gfCNCPoint1[7259] = {X 558.4447, Y 7.7679, Z -1.3333, A 0.000, B 0.000, C 0.000 }
gfCNCPoint1[7260] = {X 558.1455, Y 6.8725, Z -1.3333, A 0.000, B 0.000, C 0.000 }
gfCNCPoint1[7261] = {X 558.0443, Y 5.9339, Z -1.3333, A 0.000, B 0.000, C 0.000 }
gfCNCPoint1[7262] = {X 558.0443, Y 5.0000, Z -1.3333, A 0.000, B 0.000, C 0.000 }
gfCNCPoint1[7263] = {X 558.1353, Y 4.1097, Z -1.3333, A 0.000, B 0.000, C 0.000 }
gfCNCPoint1[7264] = {X 558.4046, Y 3.2563, Z -1.3333, A 0.000, B 0.000, C 0.000 }
gfCNCPoint1[7265] = {X 558.9155, Y 2.3718, Z -1.3333, A 0.000, B 0.000, C 0.000 }
gfCNCPoint1[7266] = {X 559.6165, Y 1.6290, Z -1.3333, A 0.000, B 0.000, C 0.000 }
gfCNCPoint1[7267] = {X 560.4700, Y 1.0678, Z -1.3333, A 0.000, B 0.000, C 0.000 }
gfCNCPoint1[7268] = {X 561.4298, Y 0.7186, Z -1.3333, A 0.000, B 0.000, C 0.000 }
gfCNCPoint1[7269] = {X 562.4443, Y 0.6000, Z -1.3333, A 0.000, B 0.000, C 0.000 }
gfCNCPoint1[7270] = {X 570.9376, Y 0.6000, Z -1.3333, A 0.000, B 0.000, C 0.000 }
gfCNCPoint1[7271] = {X 571.9521, Y 0.7186, Z -1.3333, A 0.000, B 0.000, C 0.000 }
gfCNCPoint1[7272] = {X 572.9119, Y 1.0678, Z -1.3333, A 0.000, B 0.000, C 0.000 }
gfCNCPoint1[7273] = {X 573.7653, Y 1.6290, Z -1.3333, A 0.000, B 0.000, C 0.000 }
gfCNCPoint1[7274] = {X 574.4664, Y 2.3718, Z -1.3333, A 0.000, B 0.000, C 0.000 }
gfCNCPoint1[7275] = {X 574.9773, Y 3.2563, Z -1.3333, A 0.000, B 0.000, C 0.000 }
gfCNCPoint1[7276] = {X 575.2317, Y 4.0408, Z -1.3333, A 0.000, B 0.000, C 0.000 }
gfCNCPoint1[7277] = {X 575.3353, Y 4.8590, Z -1.3333, A 0.000, B 0.000, C 0.000 }
gfCNCPoint1[7278] = {X 580.1328, Y 4.7051, Z -1.3333, A 0.000, B 0.000, C 0.000 }
gfCNCPoint1[7279] = {X 580.1364, Y 4.8525, Z -1.3333, A 0.000, B 0.000, C 0.000 }
gfCNCPoint1[7280] = {X 580.1376, Y 5.0000, Z -1.3333, A 0.000, B 0.000, C 0.000 }
gfCNCPoint1[7281] = {X 580.1376, Y 5.9338, Z -1.3333, A 0.000, B 0.000, C 0.000 }
gfCNCPoint1[7282] = {X 580.0685, Y 7.0592, Z -1.3333, A 0.000, B 0.000, C 0.000 }
gfCNCPoint1[7283] = {X 579.8623, Y 8.1677, Z -1.3333, A 0.000, B 0.000, C 0.000 }
gfCNCPoint1[7284] = {X 581.2004, Y 11.4539, Z -1.3333, A 0.000, B 0.000, C 0.000 }
gfCNCPoint1[7285] = {X 582.6186, Y 7.9855, Z -1.3333, A 0.000, B 0.000, C 0.000 }
gfCNCPoint1[7286] = {X 582.4489, Y 6.9999, Z -1.3333, A 0.000, B 0.000, C 0.000 }
gfCNCPoint1[7287] = {X 582.3872, Y 6.0018, Z -1.3333, A 0.000, B 0.000, C 0.000 }
gfCNCPoint1[7288] = {X 582.3870, Y 5.0000, Z -1.3333, A 0.000, B 0.000, C 0.000 }
gfCNCPoint1[7289] = {X 582.3881, Y 4.8525, Z -1.3333, A 0.000, B 0.000, C 0.000 }
gfCNCPoint1[7290] = {X 582.3917, Y 4.7051, Z -1.3333, A 0.000, B 0.000, C 0.000 }
gfCNCPoint1[7291] = {X 580.1328, Y 4.7051, Z -1.3333, A 0.000, B 0.000, C 0.000 }
gfCNCPoint1[7292] = {X 577.7341, Y 4.7820, Z -1.3333, A 0.000, B 0.000, C 0.000 }
gfCNCPoint1[7293] = {X 577.7367, Y 4.8910, Z -1.3333, A 0.000, B 0.000, C 0.000 }
gfCNCPoint1[7294] = {X 577.7376, Y 5.0000, Z -1.3333, A 0.000, B 0.000, C 0.000 }
gfCNCPoint1[7295] = {X 577.7376, Y 5.9339, Z -1.3333, A 0.000, B 0.000, C 0.000 }
gfCNCPoint1[7296] = {X 577.6317, Y 7.1291, Z -1.3333, A 0.000, B 0.000, C 0.000 }
gfCNCPoint1[7297] = {X 577.3175, Y 8.2871, Z -1.3333, A 0.000, B 0.000, C 0.000 }
gfCNCPoint1[7298] = {X 577.5051, Y 8.7428, Z -1.3333, A 0.000, B 0.000, C 0.000 }
gfCNCPoint1[7299] = {X 581.1958, Y 17.8065, Z -1.3333, A 0.000, B 0.000, C 0.000 }
gfCNCPoint1[7300] = {X 585.1518, Y 8.1314, Z -1.3333, A 0.000, B 0.000, C 0.000 }
gfCNCPoint1[7301] = {X 584.8835, Y 7.0761, Z -1.3333, A 0.000, B 0.000, C 0.000 }
gfCNCPoint1[7302] = {X 584.7872, Y 5.9914, Z -1.3333, A 0.000, B 0.000, C 0.000 }
gfCNCPoint1[7303] = {X 584.7870, Y 5.0000, Z -1.3333, A 0.000, B 0.000, C 0.000 }
gfCNCPoint1[7304] = {X 584.7878, Y 4.8910, Z -1.3333, A 0.000, B 0.000, C 0.000 }
gfCNCPoint1[7305] = {X 584.7904, Y 4.7820, Z -1.3333, A 0.000, B 0.000, C 0.000 }
gfCNCPoint1[7306] = {X 584.9505, Y 3.5175, Z -1.3333, A 0.000, B 0.000, C 0.000 }
gfCNCPoint1[7307] = {X 585.3438, Y 2.3051, Z -1.3333, A 0.000, B 0.000, C 0.000 }
gfCNCPoint1[7308] = {X 577.1808, Y 2.3051, Z -1.3333, A 0.000, B 0.000, C 0.000 }
gfCNCPoint1[7309] = {X 577.5740, Y 3.5175, Z -1.3333, A 0.000, B 0.000, C 0.000 }
gfCNCPoint1[7310] = {X 577.7341, Y 4.7820, Z -1.3333, A 0.000, B 0.000, C 0.000 }
gfCNCPoint1[7311] = {X 575.3353, Y 4.8590, Z -1.3333, A 0.000, B 0.000, C 0.000 }
gfCNCPoint1[7312] = {X 575.3370, Y 4.9295, Z -1.3333, A 0.000, B 0.000, C 0.000 }
gfCNCPoint1[7313] = {X 575.3376, Y 5.0000, Z -1.3333, A 0.000, B 0.000, C 0.000 }
gfCNCPoint1[7314] = {X 575.3372, Y 5.9910, Z -1.3333, A 0.000, B 0.000, C 0.000 }
gfCNCPoint1[7315] = {X 575.2576, Y 6.7693, Z -1.3333, A 0.000, B 0.000, C 0.000 }
gfCNCPoint1[7316] = {X 575.0414, Y 7.5211, Z -1.3333, A 0.000, B 0.000, C 0.000 }
gfCNCPoint1[7317] = {X 574.6954, Y 8.2228, Z -1.3333, A 0.000, B 0.000, C 0.000 }
gfCNCPoint1[7318] = {X 575.2866, Y 9.6583, Z -1.3333, A 0.000, B 0.000, C 0.000 }
gfCNCPoint1[7319] = {X 578.9730, Y 18.7116, Z -1.3333, A 0.000, B 0.000, C 0.000 }
gfCNCPoint1[7320] = {X 580.9325, Y 23.5237, Z -1.3333, A 0.000, B 0.000, C 0.000 }
gfCNCPoint1[7321] = {X 581.1912, Y 24.1591, Z -1.3333, A 0.000, B 0.000, C 0.000 }
gfCNCPoint1[7322] = {X 587.7573, Y 8.1005, Z -1.3333, A 0.000, B 0.000, C 0.000 }
gfCNCPoint1[7323] = {X 587.4436, Y 7.4147, Z -1.3333, A 0.000, B 0.000, C 0.000 }
gfCNCPoint1[7324] = {X 587.2516, Y 6.6853, Z -1.3333, A 0.000, B 0.000, C 0.000 }
gfCNCPoint1[7325] = {X 587.1870, Y 5.9339, Z -1.3333, A 0.000, B 0.000, C 0.000 }
gfCNCPoint1[7326] = {X 587.1870, Y 5.0000, Z -1.3333, A 0.000, B 0.000, C 0.000 }
gfCNCPoint1[7327] = {X 587.2780, Y 4.1097, Z -1.3333, A 0.000, B 0.000, C 0.000 }
gfCNCPoint1[7328] = {X 587.5472, Y 3.2563, Z -1.3333, A 0.000, B 0.000, C 0.000 }
gfCNCPoint1[7329] = {X 588.0581, Y 2.3718, Z -1.3333, A 0.000, B 0.000, C 0.000 }
gfCNCPoint1[7330] = {X 588.7592, Y 1.6290, Z -1.3333, A 0.000, B 0.000, C 0.000 }
gfCNCPoint1[7331] = {X 589.6126, Y 1.0678, Z -1.3333, A 0.000, B 0.000, C 0.000 }
gfCNCPoint1[7332] = {X 590.5725, Y 0.7186, Z -1.3333, A 0.000, B 0.000, C 0.000 }
gfCNCPoint1[7333] = {X 591.5870, Y 0.6000, Z -1.3333, A 0.000, B 0.000, C 0.000 }
gfCNCPoint1[7334] = {X 600.0000, Y 0.6000, Z -1.3333, A 0.000, B 0.000, C 0.000 }
gfCNCPoint1[7335] = {X 600.8720, Y 0.6873, Z -1.3333, A 0.000, B 0.000, C 0.000 }
gfCNCPoint1[7336] = {X 601.7093, Y 0.9456, Z -1.3333, A 0.000, B 0.000, C 0.000 }
gfCNCPoint1[7337] = {X 602.4789, Y 1.3648, Z -1.3333, A 0.000, B 0.000, C 0.000 }
gfCNCPoint1[7338] = {X 603.1502, Y 1.9281, Z -1.3333, A 0.000, B 0.000, C 0.000 }
gfCNCPoint1[7339] = {X 603.6965, Y 2.6133, Z -1.3333, A 0.000, B 0.000, C 0.000 }
gfCNCPoint1[7340] = {X 603.6965, Y 1.8140, Z -1.3333, A 0.000, B 0.000, C 0.000 }
gfCNCPoint1[7341] = {X 602.9511, Y 1.1135, Z -1.3333, A 0.000, B 0.000, C 0.000 }
gfCNCPoint1[7342] = {X 602.0762, Y 0.5837, Z -1.3333, A 0.000, B 0.000, C 0.000 }
gfCNCPoint1[7343] = {X 601.1100, Y 0.2479, Z -1.3333, A 0.000, B 0.000, C 0.000 }
gfCNCPoint1[7344] = {X 600.0950, Y 0.1209, Z -1.3333, A 0.000, B 0.000, C 0.000 }
gfCNCPoint1[7345] = {X 600.0947, Y -0.0187, Z -1.3333, A 0.000, B 0.000, C 0.000 }
gfCNCPoint1[7346] = {X 600.0671, Y -0.0697, Z -1.3333, A 0.000, B 0.000, C 0.000 }
gfCNCPoint1[7347] = {X 600.0148, Y -0.0949, Z -1.3333, A 0.000, B 0.000, C 0.000 }
gfCNCPoint1[7348] = {X 351.5614, Y -0.0949, Z -1.3333, A 0.000, B 0.000, C 0.000 }
gfCNCPoint1[7349] = {X 351.4045, Y -0.1238, Z -1.3333, A 0.000, B 0.000, C 0.000 }
gfCNCPoint1[7350] = {X 348.9100, Y -0.4700, Z -1.3333, A 0.000, B 0.000, C 0.000 }
gfCNCPoint1[7351] = {X 346.3941, Y -0.5809, Z -1.3333, A 0.000, B 0.000, C 0.000 }
gfCNCPoint1[7352] = {X 343.8788, Y -0.4555, Z -1.3333, A 0.000, B 0.000, C 0.000 }
gfCNCPoint1[7353] = {X 341.3863, Y -0.0949, Z -1.3333, A 0.000, B 0.000, C 0.000 }
gfCNCPoint1[7354] = {X -0.0148, Y -0.0949, Z -1.3333, A 0.000, B 0.000, C 0.000 }
gfCNCPoint1[7355] = {X -0.0671, Y -0.0697, Z -1.3333, A 0.000, B 0.000, C 0.000 }
gfCNCPoint1[7356] = {X -0.0947, Y -0.0187, Z -1.3333, A 0.000, B 0.000, C 0.000 }
gfCNCPoint1[7357] = {X -0.0965, Y 0.8569, Z -1.3333, A 0.000, B 0.000, C 0.000 }
gfCNCPoint1[7358] = {X -0.0965, Y 8.7890, Z -1.3333, A 0.000, B 0.000, C 0.000 }
gfCNCPoint1[7359] = {X -0.7633, Y 8.9979, Z -1.3333, A 0.000, B 0.000, C 0.000 }
gfCNCPoint1[7360] = {X -1.3935, Y 9.2998, Z -1.3333, A 0.000, B 0.000, C 0.000 }
gfCNCPoint1[7361] = {X -1.9904, Y 9.6404, Z -1.3333, A 0.000, B 0.000, C 0.000 }
gfCNCPoint1[7362] = {X -2.6454, Y 10.0884, Z -1.3333, A 0.000, B 0.000, C 0.000 }
gfCNCPoint1[7363] = {X -3.2192, Y 10.6366, Z -1.3333, A 0.000, B 0.000, C 0.000 }
gfCNCPoint1[7364] = {X -3.6965, Y 11.2705, Z -1.3333, A 0.000, B 0.000, C 0.000 }
gfCNCPoint1[7365] = {X -3.6965, Y 12.3459, Z -1.3333, A 0.000, B 0.000, C 0.000 }
gfCNCPoint1[7366] = {X -3.2331, Y 11.4382, Z -1.3333, A 0.000, B 0.000, C 0.000 }
gfCNCPoint1[7367] = {X -2.5733, Y 10.6615, Z -1.3333, A 0.000, B 0.000, C 0.000 }
gfCNCPoint1[7368] = {X -1.7526, Y 10.0573, Z -1.3333, A 0.000, B 0.000, C 0.000 }
gfCNCPoint1[7369] = {X -1.0994, Y 9.6852, Z -1.3333, A 0.000, B 0.000, C 0.000 }
gfCNCPoint1[7370] = {X -0.1607, Y 9.3012, Z -1.3333, A 0.000, B 0.000, C 0.000 }
gfCNCPoint1[7371] = {X 0.8409, Y 9.1423, Z -1.3333, A 0.000, B 0.000, C 0.000 }
gfCNCPoint1[7372] = {X 1.8523, Y 9.2169, Z -1.3333, A 0.000, B 0.000, C 0.000 }
gfCNCPoint1[7373] = {X 2.2372, Y 9.3088, Z -1.3333, A 0.000, B 0.000, C 0.000 }
gfCNCPoint1[7374] = {X 2.6123, Y 9.4348, Z -1.3333, A 0.000, B 0.000, C 0.000 }
gfCNCPoint1[7375] = {X 3.3801, Y 9.0795, Z -1.3333, A 0.000, B 0.000, C 0.000 }
gfCNCPoint1[7376] = {X 4.1677, Y 8.7704, Z -1.3333, A 0.000, B 0.000, C 0.000 }
gfCNCPoint1[7377] = {X 6.0851, Y 8.0995, Z -1.3333, A 0.000, B 0.000, C 0.000 }
gfCNCPoint1[7378] = {X 8.0532, Y 7.5963, Z -1.3333, A 0.000, B 0.000, C 0.000 }
gfCNCPoint1[7379] = {X 10.0574, Y 7.2648, Z -1.3333, A 0.000, B 0.000, C 0.000 }
gfCNCPoint1[7380] = {X 12.0827, Y 7.1073, Z -1.3333, A 0.000, B 0.000, C 0.000 }
gfCNCPoint1[7381] = {X 14.1141, Y 7.1249, Z -1.3333, A 0.000, B 0.000, C 0.000 }
gfCNCPoint1[7382] = {X 16.1363, Y 7.3177, Z -1.3333, A 0.000, B 0.000, C 0.000 }
gfCNCPoint1[7383] = {X 16.5409, Y 7.3732, Z -1.3333, A 0.000, B 0.000, C 0.000 }
gfCNCPoint1[7384] = {X 18.2850, Y 7.7308, Z -1.3333, A 0.000, B 0.000, C 0.000 }
gfCNCPoint1[7385] = {X 19.9840, Y 8.2634, Z -1.3333, A 0.000, B 0.000, C 0.000 }
gfCNCPoint1[7386] = {X 21.6202, Y 8.9655, Z -1.3333, A 0.000, B 0.000, C 0.000 }
gfCNCPoint1[7387] = {X 23.1768, Y 9.8298, Z -1.3333, A 0.000, B 0.000, C 0.000 }
gfCNCPoint1[7388] = {X 24.6377, Y 10.8475, Z -1.3333, A 0.000, B 0.000, C 0.000 }
gfCNCPoint1[7389] = {X 25.7295, Y 11.8031, Z -1.3333, A 0.000, B 0.000, C 0.000 }
gfCNCPoint1[7390] = {X 26.7088, Y 12.8735, Z -1.3333, A 0.000, B 0.000, C 0.000 }
gfCNCPoint1[7391] = {X 27.5636, Y 14.0458, Z -1.3333, A 0.000, B 0.000, C 0.000 }
gfCNCPoint1[7392] = {X 28.2836, Y 15.3054, Z -1.3333, A 0.000, B 0.000, C 0.000 }
gfCNCPoint1[7393] = {X 28.8598, Y 16.6369, Z -1.3333, A 0.000, B 0.000, C 0.000 }
gfCNCPoint1[7394] = {X 29.3358, Y 18.3014, Z -1.3333, A 0.000, B 0.000, C 0.000 }
gfCNCPoint1[7395] = {X 29.6183, Y 20.0095, Z -1.3333, A 0.000, B 0.000, C 0.000 }
gfCNCPoint1[7396] = {X 29.7035, Y 21.7387, Z -1.3333, A 0.000, B 0.000, C 0.000 }
gfCNCPoint1[7397] = {X 29.5903, Y 23.4663, Z -1.3333, A 0.000, B 0.000, C 0.000 }
gfCNCPoint1[7398] = {X 29.2802, Y 25.1696, Z -1.3333, A 0.000, B 0.000, C 0.000 }
gfCNCPoint1[7399] = {X 28.7891, Y 26.7453, Z -1.3333, A 0.000, B 0.000, C 0.000 }
gfCNCPoint1[7400] = {X 28.0825, Y 28.2367, Z -1.3333, A 0.000, B 0.000, C 0.000 }
gfCNCPoint1[7401] = {X 27.1741, Y 29.6147, Z -1.3333, A 0.000, B 0.000, C 0.000 }
gfCNCPoint1[7402] = {X 26.3570, Y 30.5719, Z -1.3333, A 0.000, B 0.000, C 0.000 }
gfCNCPoint1[7403] = {X 25.4424, Y 31.4364, Z -1.3333, A 0.000, B 0.000, C 0.000 }
gfCNCPoint1[7404] = {X 25.6930, Y 31.5320, Z -1.3333, A 0.000, B 0.000, C 0.000 }
gfCNCPoint1[7405] = {X 25.9374, Y 31.6427, Z -1.3333, A 0.000, B 0.000, C 0.000 }
gfCNCPoint1[7406] = {X 26.6622, Y 32.0899, Z -1.3333, A 0.000, B 0.000, C 0.000 }
gfCNCPoint1[7407] = {X 27.2873, Y 32.6684, Z -1.3333, A 0.000, B 0.000, C 0.000 }
gfCNCPoint1[7408] = {X 27.6590, Y 33.1492, Z -1.3333, A 0.000, B 0.000, C 0.000 }
gfCNCPoint1[7409] = {X 27.9609, Y 33.6766, Z -1.3333, A 0.000, B 0.000, C 0.000 }
gfCNCPoint1[7410] = {X 30.9820, Y 39.9182, Z -1.3333, A 0.000, B 0.000, C 0.000 }
gfCNCPoint1[7411] = {X 31.3085, Y 40.8441, Z -1.3333, A 0.000, B 0.000, C 0.000 }
gfCNCPoint1[7412] = {X 31.4215, Y 41.8194, Z -1.3333, A 0.000, B 0.000, C 0.000 }
gfCNCPoint1[7413] = {X 31.3155, Y 42.7955, Z -1.3333, A 0.000, B 0.000, C 0.000 }
gfCNCPoint1[7414] = {X 30.9956, Y 43.7238, Z -1.3333, A 0.000, B 0.000, C 0.000 }
gfCNCPoint1[7415] = {X 30.4779, Y 44.5580, Z -1.3333, A 0.000, B 0.000, C 0.000 }
gfCNCPoint1[7416] = {X 29.7880, Y 45.2567, Z -1.3333, A 0.000, B 0.000, C 0.000 }
gfCNCPoint1[7417] = {X 29.2515, Y 45.6905, Z -1.3333, A 0.000, B 0.000, C 0.000 }
gfCNCPoint1[7418] = {X 28.5397, Y 46.1587, Z -1.3333, A 0.000, B 0.000, C 0.000 }
gfCNCPoint1[7419] = {X 27.7513, Y 46.4816, Z -1.3333, A 0.000, B 0.000, C 0.000 }
gfCNCPoint1[7420] = {X 26.9155, Y 46.6472, Z -1.3333, A 0.000, B 0.000, C 0.000 }
gfCNCPoint1[7421] = {X 26.0635, Y 46.6494, Z -1.3333, A 0.000, B 0.000, C 0.000 }
gfCNCPoint1[7422] = {X 25.2269, Y 46.4880, Z -1.3333, A 0.000, B 0.000, C 0.000 }
gfCNCPoint1[7423] = {X 23.2106, Y 47.5426, Z -1.3333, A 0.000, B 0.000, C 0.000 }
gfCNCPoint1[7424] = {X 21.1166, Y 48.4331, Z -1.3333, A 0.000, B 0.000, C 0.000 }
gfCNCPoint1[7425] = {X 18.9583, Y 49.1538, Z -1.3333, A 0.000, B 0.000, C 0.000 }
gfCNCPoint1[7426] = {X 18.4672, Y 49.2899, Z -1.3333, A 0.000, B 0.000, C 0.000 }
gfCNCPoint1[7427] = {X 16.5967, Y 49.7226, Z -1.3333, A 0.000, B 0.000, C 0.000 }
gfCNCPoint1[7428] = {X 14.6960, Y 49.9931, Z -1.3333, A 0.000, B 0.000, C 0.000 }
gfCNCPoint1[7429] = {X 12.7791, Y 50.0995, Z -1.3333, A 0.000, B 0.000, C 0.000 }
gfCNCPoint1[7430] = {X 10.8601, Y 50.0409, Z -1.3333, A 0.000, B 0.000, C 0.000 }
gfCNCPoint1[7431] = {X 8.9532, Y 49.8178, Z -1.3333, A 0.000, B 0.000, C 0.000 }
gfCNCPoint1[7432] = {X 8.2283, Y 49.7011, Z -1.3333, A 0.000, B 0.000, C 0.000 }
gfCNCPoint1[7433] = {X 6.5700, Y 49.3105, Z -1.3333, A 0.000, B 0.000, C 0.000 }
gfCNCPoint1[7434] = {X 4.9585, Y 48.7578, Z -1.3333, A 0.000, B 0.000, C 0.000 }
gfCNCPoint1[7435] = {X 3.4094, Y 48.0486, Z -1.3333, A 0.000, B 0.000, C 0.000 }
gfCNCPoint1[7436] = {X 2.3355, Y 47.4411, Z -1.3333, A 0.000, B 0.000, C 0.000 }
gfCNCPoint1[7437] = {X 1.3077, Y 46.7583, Z -1.3333, A 0.000, B 0.000, C 0.000 }
gfCNCPoint1[7438] = {X -0.0256, Y 45.6860, Z -1.3333, A 0.000, B 0.000, C 0.000 }
gfCNCPoint1[7439] = {X -1.2107, Y 44.4520, Z -1.3333, A 0.000, B 0.000, C 0.000 }
gfCNCPoint1[7440] = {X -2.2282, Y 43.0765, Z -1.3333, A 0.000, B 0.000, C 0.000 }
gfCNCPoint1[7441] = {X -3.0614, Y 41.5820, Z -1.3333, A 0.000, B 0.000, C 0.000 }
gfCNCPoint1[7442] = {X -3.6965, Y 39.9933, Z -1.3333, A 0.000, B 0.000, C 0.000 }
gfCNCPoint1[7443] = {X -3.6965, Y 41.3449, Z -1.3333, A 0.000, B 0.000, C 0.000 }
gfCNCPoint1[7444] = {X -3.0079, Y 42.7182, Z -1.3333, A 0.000, B 0.000, C 0.000 }
gfCNCPoint1[7445] = {X -2.1712, Y 44.0066, Z -1.3333, A 0.000, B 0.000, C 0.000 }
gfCNCPoint1[7446] = {X -1.1967, Y 45.1942, Z -1.3333, A 0.000, B 0.000, C 0.000 }
gfCNCPoint1[7447] = {X -0.0965, Y 46.2663, Z -1.3333, A 0.000, B 0.000, C 0.000 }
gfCNCPoint1[7448] = {X -0.0965, Y 99.1431, Z -1.3333, A 0.000, B 0.000, C 0.000 }
gfCNCPoint1[7449] = {X -0.0947, Y 100.0187, Z -1.3333, A 0.000, B 0.000, C 0.000 }
gfCNCPoint1[7450] = {X -0.0671, Y 100.0697, Z -1.3333, A 0.000, B 0.000, C 0.000 }
gfCNCPoint1[7451] = {X -0.0148, Y 100.0949, Z -1.3333, A 0.000, B 0.000, C 0.000 }
gfCNCPoint1[7452] = {X 120.5925, Y 100.0949, Z -1.3333, A 0.000, B 0.000, C 0.000 }
gfCNCPoint1[7453] = {X 121.0613, Y 100.8811, Z -1.3333, A 0.000, B 0.000, C 0.000 }
gfCNCPoint1[7454] = {X 121.6686, Y 101.5660, Z -1.3333, A 0.000, B 0.000, C 0.000 }
gfCNCPoint1[7455] = {X 122.3931, Y 102.1254, Z -1.3333, A 0.000, B 0.000, C 0.000 }
gfCNCPoint1[7456] = {X 123.2094, Y 102.5396, Z -1.3333, A 0.000, B 0.000, C 0.000 }
gfCNCPoint1[7457] = {X 124.0887, Y 102.7942, Z -1.3333, A 0.000, B 0.000, C 0.000 }
gfCNCPoint1[7458] = {X 125.0000, Y 102.8800, Z -1.3333, A 0.000, B 0.000, C 0.000 }
gfCNCPoint1[7459] = {X 143.7791, Y 102.8800, Z -1.3333, A 0.000, B 0.000, C 0.000 }
gfCNCPoint1[7460] = {X 144.6904, Y 102.7942, Z -1.3333, A 0.000, B 0.000, C 0.000 }
gfCNCPoint1[7461] = {X 145.5697, Y 102.5396, Z -1.3333, A 0.000, B 0.000, C 0.000 }
gfCNCPoint1[7462] = {X 146.3860, Y 102.1254, Z -1.3333, A 0.000, B 0.000, C 0.000 }
gfCNCPoint1[7463] = {X 147.1105, Y 101.5660, Z -1.3333, A 0.000, B 0.000, C 0.000 }
gfCNCPoint1[7464] = {X 147.7178, Y 100.8811, Z -1.3333, A 0.000, B 0.000, C 0.000 }
gfCNCPoint1[7465] = {X 148.1866, Y 100.0949, Z -1.3333, A 0.000, B 0.000, C 0.000 }
gfCNCPoint1[7466] = {X 150.8370, Y 100.0949, Z -1.3333, A 0.000, B 0.000, C 0.000 }
gfCNCPoint1[7467] = {X 150.8370, Y 95.2949, Z -1.3333, A 0.000, B 0.000, C 0.000 }
gfCNCPoint1[7468] = {X 187.9257, Y 95.2949, Z -1.3333, A 0.000, B 0.000, C 0.000 }
gfCNCPoint1[7469] = {X 187.9777, Y 95.0989, Z -1.3333, A 0.000, B 0.000, C 0.000 }
gfCNCPoint1[7470] = {X 188.0352, Y 94.9045, Z -1.3333, A 0.000, B 0.000, C 0.000 }
gfCNCPoint1[7471] = {X 187.2619, Y 94.0602, Z -1.3333, A 0.000, B 0.000, C 0.000 }
gfCNCPoint1[7472] = {X 151.4055, Y 94.0602, Z -1.3333, A 0.000, B 0.000, C 0.000 }
gfCNCPoint1[7473] = {X 150.7052, Y 94.8361, Z -1.3333, A 0.000, B 0.000, C 0.000 }
gfCNCPoint1[7474] = {X 150.7748, Y 95.0644, Z -1.3333, A 0.000, B 0.000, C 0.000 }
gfCNCPoint1[7475] = {X 150.8370, Y 95.2949, Z -1.3333, A 0.000, B 0.000, C 0.000 }
gfCNCPoint1[7476] = {X 150.8370, Y 97.6949, Z -1.3333, A 0.000, B 0.000, C 0.000 }
gfCNCPoint1[7477] = {X 190.1070, Y 97.6949, Z -1.3333, A 0.000, B 0.000, C 0.000 }
gfCNCPoint1[7478] = {X 190.1070, Y 97.0659, Z -1.3333, A 0.000, B 0.000, C 0.000 }
gfCNCPoint1[7479] = {X 190.1938, Y 96.1495, Z -1.3333, A 0.000, B 0.000, C 0.000 }
gfCNCPoint1[7480] = {X 190.4511, Y 95.2657, Z -1.3333, A 0.000, B 0.000, C 0.000 }
gfCNCPoint1[7481] = {X 190.8699, Y 94.4460, Z -1.3333, A 0.000, B 0.000, C 0.000 }
gfCNCPoint1[7482] = {X 188.3182, Y 91.6602, Z -1.3333, A 0.000, B 0.000, C 0.000 }
gfCNCPoint1[7483] = {X 150.3387, Y 91.6602, Z -1.3333, A 0.000, B 0.000, C 0.000 }
gfCNCPoint1[7484] = {X 147.8631, Y 94.4029, Z -1.3333, A 0.000, B 0.000, C 0.000 }
gfCNCPoint1[7485] = {X 148.2972, Y 95.2330, Z -1.3333, A 0.000, B 0.000, C 0.000 }
gfCNCPoint1[7486] = {X 148.5657, Y 96.1303, Z -1.3333, A 0.000, B 0.000, C 0.000 }
gfCNCPoint1[7487] = {X 148.6591, Y 97.0623, Z -1.3333, A 0.000, B 0.000, C 0.000 }
gfCNCPoint1[7488] = {X 148.6591, Y 97.6949, Z -1.3333, A 0.000, B 0.000, C 0.000 }
gfCNCPoint1[7489] = {X 150.8370, Y 97.6949, Z -1.3333, A 0.000, B 0.000, C 0.000 }
gfCNCPoint1[7490] = {X 150.8370, Y 100.0949, Z -1.3333, A 0.000, B 0.000, C 0.000 }
gfCNCPoint1[7491] = {X 190.5795, Y 100.0949, Z -1.3333, A 0.000, B 0.000, C 0.000 }
gfCNCPoint1[7492] = {X 191.0482, Y 100.8811, Z -1.3333, A 0.000, B 0.000, C 0.000 }
gfCNCPoint1[7493] = {X 191.6556, Y 101.5660, Z -1.3333, A 0.000, B 0.000, C 0.000 }
gfCNCPoint1[7494] = {X 192.3801, Y 102.1254, Z -1.3333, A 0.000, B 0.000, C 0.000 }
gfCNCPoint1[7495] = {X 193.1964, Y 102.5396, Z -1.3333, A 0.000, B 0.000, C 0.000 }
gfCNCPoint1[7496] = {X 194.0756, Y 102.7942, Z -1.3333, A 0.000, B 0.000, C 0.000 }
gfCNCPoint1[7497] = {X 194.9870, Y 102.8800, Z -1.3333, A 0.000, B 0.000, C 0.000 }
gfCNCPoint1[7498] = {X 212.6141, Y 102.8800, Z -1.3333, A 0.000, B 0.000, C 0.000 }
gfCNCPoint1[7499] = {X 213.0066, Y 102.8642, Z -1.3333, A 0.000, B 0.000, C 0.000 }
gfCNCPoint1[7500] = {X 213.3966, Y 102.8169, Z -1.3333, A 0.000, B 0.000, C 0.000 }
gfCNCPoint1[7501] = {X 213.7865, Y 102.8642, Z -1.3333, A 0.000, B 0.000, C 0.000 }
gfCNCPoint1[7502] = {X 214.1790, Y 102.8800, Z -1.3333, A 0.000, B 0.000, C 0.000 }
gfCNCPoint1[7503] = {X 233.4798, Y 102.8800, Z -1.3333, A 0.000, B 0.000, C 0.000 }
gfCNCPoint1[7504] = {X 234.3911, Y 102.7942, Z -1.3333, A 0.000, B 0.000, C 0.000 }
gfCNCPoint1[7505] = {X 235.2704, Y 102.5396, Z -1.3333, A 0.000, B 0.000, C 0.000 }
gfCNCPoint1[7506] = {X 236.0866, Y 102.1254, Z -1.3333, A 0.000, B 0.000, C 0.000 }
gfCNCPoint1[7507] = {X 236.8112, Y 101.5660, Z -1.3333, A 0.000, B 0.000, C 0.000 }
gfCNCPoint1[7508] = {X 237.4185, Y 100.8811, Z -1.3333, A 0.000, B 0.000, C 0.000 }
gfCNCPoint1[7509] = {X 237.8873, Y 100.0949, Z -1.3333, A 0.000, B 0.000, C 0.000 }
gfCNCPoint1[7510] = {X 261.4765, Y 100.0949, Z -1.3333, A 0.000, B 0.000, C 0.000 }
gfCNCPoint1[7511] = {X 261.4765, Y 90.4949, Z -1.3333, A 0.000, B 0.000, C 0.000 }
gfCNCPoint1[7512] = {X 266.0962, Y 90.4949, Z -1.3333, A 0.000, B 0.000, C 0.000 }
gfCNCPoint1[7513] = {X 266.1752, Y 90.3746, Z -1.3333, A 0.000, B 0.000, C 0.000 }
gfCNCPoint1[7514] = {X 266.2556, Y 90.2554, Z -1.3333, A 0.000, B 0.000, C 0.000 }
gfCNCPoint1[7515] = {X 263.5087, Y 89.1786, Z -1.3333, A 0.000, B 0.000, C 0.000 }
gfCNCPoint1[7516] = {X 261.4765, Y 90.4949, Z -1.3333, A 0.000, B 0.000, C 0.000 }
gfCNCPoint1[7517] = {X 261.4765, Y 92.8949, Z -1.3333, A 0.000, B 0.000, C 0.000 }
gfCNCPoint1[7518] = {X 267.4974, Y 92.8949, Z -1.3333, A 0.000, B 0.000, C 0.000 }
gfCNCPoint1[7519] = {X 267.8429, Y 92.2375, Z -1.3333, A 0.000, B 0.000, C 0.000 }
gfCNCPoint1[7520] = {X 268.2378, Y 91.6085, Z -1.3333, A 0.000, B 0.000, C 0.000 }
gfCNCPoint1[7521] = {X 269.1700, Y 90.4463, Z -1.3333, A 0.000, B 0.000, C 0.000 }
gfCNCPoint1[7522] = {X 270.2694, Y 89.4409, Z -1.3333, A 0.000, B 0.000, C 0.000 }
gfCNCPoint1[7523] = {X 270.2694, Y 89.2510, Z -1.3333, A 0.000, B 0.000, C 0.000 }
gfCNCPoint1[7524] = {X 263.2378, Y 86.4946, Z -1.3333, A 0.000, B 0.000, C 0.000 }
gfCNCPoint1[7525] = {X 253.3566, Y 92.8949, Z -1.3333, A 0.000, B 0.000, C 0.000 }
gfCNCPoint1[7526] = {X 261.4765, Y 92.8949, Z -1.3333, A 0.000, B 0.000, C 0.000 }
gfCNCPoint1[7527] = {X 261.4765, Y 95.2949, Z -1.3333, A 0.000, B 0.000, C 0.000 }
gfCNCPoint1[7528] = {X 269.1714, Y 95.2949, Z -1.3333, A 0.000, B 0.000, C 0.000 }
gfCNCPoint1[7529] = {X 269.5516, Y 94.1744, Z -1.3333, A 0.000, B 0.000, C 0.000 }
gfCNCPoint1[7530] = {X 270.1083, Y 93.1302, Z -1.3333, A 0.000, B 0.000, C 0.000 }
gfCNCPoint1[7531] = {X 270.8267, Y 92.1901, Z -1.3333, A 0.000, B 0.000, C 0.000 }
gfCNCPoint1[7532] = {X 271.6880, Y 91.3787, Z -1.3333, A 0.000, B 0.000, C 0.000 }
gfCNCPoint1[7533] = {X 272.6694, Y 90.7176, Z -1.3333, A 0.000, B 0.000, C 0.000 }
gfCNCPoint1[7534] = {X 272.6694, Y 87.6139, Z -1.3333, A 0.000, B 0.000, C 0.000 }
gfCNCPoint1[7535] = {X 262.9669, Y 83.8106, Z -1.3333, A 0.000, B 0.000, C 0.000 }
gfCNCPoint1[7536] = {X 245.2366, Y 95.2949, Z -1.3333, A 0.000, B 0.000, C 0.000 }
gfCNCPoint1[7537] = {X 261.4765, Y 95.2949, Z -1.3333, A 0.000, B 0.000, C 0.000 }
gfCNCPoint1[7538] = {X 261.4765, Y 97.6949, Z -1.3333, A 0.000, B 0.000, C 0.000 }
gfCNCPoint1[7539] = {X 271.3527, Y 97.6949, Z -1.3333, A 0.000, B 0.000, C 0.000 }
gfCNCPoint1[7540] = {X 271.3529, Y 97.0186, Z -1.3333, A 0.000, B 0.000, C 0.000 }
gfCNCPoint1[7541] = {X 271.4810, Y 95.9545, Z -1.3333, A 0.000, B 0.000, C 0.000 }
gfCNCPoint1[7542] = {X 271.8382, Y 94.9440, Z -1.3333, A 0.000, B 0.000, C 0.000 }
gfCNCPoint1[7543] = {X 272.4073, Y 94.0359, Z -1.3333, A 0.000, B 0.000, C 0.000 }
gfCNCPoint1[7544] = {X 273.1610, Y 93.2739, Z -1.3333, A 0.000, B 0.000, C 0.000 }
gfCNCPoint1[7545] = {X 274.0629, Y 92.6949, Z -1.3333, A 0.000, B 0.000, C 0.000 }
gfCNCPoint1[7546] = {X 275.0694, Y 92.3266, Z -1.3333, A 0.000, B 0.000, C 0.000 }
gfCNCPoint1[7547] = {X 275.0694, Y 85.9769, Z -1.3333, A 0.000, B 0.000, C 0.000 }
gfCNCPoint1[7548] = {X 262.6982, Y 81.1274, Z -1.3333, A 0.000, B 0.000, C 0.000 }
gfCNCPoint1[7549] = {X 262.5768, Y 81.2038, Z -1.3333, A 0.000, B 0.000, C 0.000 }
gfCNCPoint1[7550] = {X 238.3583, Y 96.8907, Z -1.3333, A 0.000, B 0.000, C 0.000 }
gfCNCPoint1[7551] = {X 238.3598, Y 97.0659, Z -1.3333, A 0.000, B 0.000, C 0.000 }
gfCNCPoint1[7552] = {X 238.3598, Y 97.6949, Z -1.3333, A 0.000, B 0.000, C 0.000 }
gfCNCPoint1[7553] = {X 261.4765, Y 97.6949, Z -1.3333, A 0.000, B 0.000, C 0.000 }
gfCNCPoint1[7554] = {X 261.4765, Y 100.0949, Z -1.3333, A 0.000, B 0.000, C 0.000 }
gfCNCPoint1[7555] = {X 271.8252, Y 100.0949, Z -1.3333, A 0.000, B 0.000, C 0.000 }
gfCNCPoint1[7556] = {X 272.2940, Y 100.8811, Z -1.3333, A 0.000, B 0.000, C 0.000 }
gfCNCPoint1[7557] = {X 272.9013, Y 101.5660, Z -1.3333, A 0.000, B 0.000, C 0.000 }
gfCNCPoint1[7558] = {X 273.6258, Y 102.1254, Z -1.3333, A 0.000, B 0.000, C 0.000 }
gfCNCPoint1[7559] = {X 274.4421, Y 102.5396, Z -1.3333, A 0.000, B 0.000, C 0.000 }
gfCNCPoint1[7560] = {X 275.3214, Y 102.7942, Z -1.3333, A 0.000, B 0.000, C 0.000 }
gfCNCPoint1[7561] = {X 276.2327, Y 102.8800, Z -1.3333, A 0.000, B 0.000, C 0.000 }
gfCNCPoint1[7562] = {X 292.7731, Y 102.8800, Z -1.3333, A 0.000, B 0.000, C 0.000 }
gfCNCPoint1[7563] = {X 293.6844, Y 102.7942, Z -1.3333, A 0.000, B 0.000, C 0.000 }
gfCNCPoint1[7564] = {X 294.5637, Y 102.5396, Z -1.3333, A 0.000, B 0.000, C 0.000 }
gfCNCPoint1[7565] = {X 295.3799, Y 102.1254, Z -1.3333, A 0.000, B 0.000, C 0.000 }
gfCNCPoint1[7566] = {X 296.1045, Y 101.5660, Z -1.3333, A 0.000, B 0.000, C 0.000 }
gfCNCPoint1[7567] = {X 296.7118, Y 100.8811, Z -1.3333, A 0.000, B 0.000, C 0.000 }
gfCNCPoint1[7568] = {X 297.1806, Y 100.0949, Z -1.3333, A 0.000, B 0.000, C 0.000 }
gfCNCPoint1[7569] = {X 319.1370, Y 100.0949, Z -1.3333, A 0.000, B 0.000, C 0.000 }
gfCNCPoint1[7570] = {X 321.4387, Y 100.8673, Z -1.3333, A 0.000, B 0.000, C 0.000 }
gfCNCPoint1[7571] = {X 323.7830, Y 101.4988, Z -1.3333, A 0.000, B 0.000, C 0.000 }
gfCNCPoint1[7572] = {X 326.1613, Y 101.9871, Z -1.3333, A 0.000, B 0.000, C 0.000 }
gfCNCPoint1[7573] = {X 329.6396, Y 102.5406, Z -1.3333, A 0.000, B 0.000, C 0.000 }
gfCNCPoint1[7574] = {X 333.1371, Y 102.9560, Z -1.3333, A 0.000, B 0.000, C 0.000 }
gfCNCPoint1[7575] = {X 336.6483, Y 103.2328, Z -1.3333, A 0.000, B 0.000, C 0.000 }
gfCNCPoint1[7576] = {X 342.8092, Y 103.5147, Z -1.3333, A 0.000, B 0.000, C 0.000 }
gfCNCPoint1[7577] = {X 348.9761, Y 103.5913, Z -1.3333, A 0.000, B 0.000, C 0.000 }
gfCNCPoint1[7578] = {X 355.1421, Y 103.4625, Z -1.3333, A 0.000, B 0.000, C 0.000 }
gfCNCPoint1[7579] = {X 361.3005, Y 103.1283, Z -1.3333, A 0.000, B 0.000, C 0.000 }
gfCNCPoint1[7580] = {X 365.1926, Y 102.7577, Z -1.3333, A 0.000, B 0.000, C 0.000 }
gfCNCPoint1[7581] = {X 369.0624, Y 102.2005, Z -1.3333, A 0.000, B 0.000, C 0.000 }
gfCNCPoint1[7582] = {X 372.9009, Y 101.4578, Z -1.3333, A 0.000, B 0.000, C 0.000 }
gfCNCPoint1[7583] = {X 375.2305, Y 100.8566, Z -1.3333, A 0.000, B 0.000, C 0.000 }
gfCNCPoint1[7584] = {X 377.5126, Y 100.0949, Z -1.3333, A 0.000, B 0.000, C 0.000 }
gfCNCPoint1[7585] = {X 391.9985, Y 100.0949, Z -1.3333, A 0.000, B 0.000, C 0.000 }
gfCNCPoint1[7586] = {X 392.4672, Y 100.8811, Z -1.3333, A 0.000, B 0.000, C 0.000 }
gfCNCPoint1[7587] = {X 393.0746, Y 101.5660, Z -1.3333, A 0.000, B 0.000, C 0.000 }
gfCNCPoint1[7588] = {X 393.7991, Y 102.1254, Z -1.3333, A 0.000, B 0.000, C 0.000 }
gfCNCPoint1[7589] = {X 394.6154, Y 102.5396, Z -1.3333, A 0.000, B 0.000, C 0.000 }
gfCNCPoint1[7590] = {X 395.4946, Y 102.7942, Z -1.3333, A 0.000, B 0.000, C 0.000 }
gfCNCPoint1[7591] = {X 396.4059, Y 102.8800, Z -1.3333, A 0.000, B 0.000, C 0.000 }
gfCNCPoint1[7592] = {X 415.7067, Y 102.8800, Z -1.3333, A 0.000, B 0.000, C 0.000 }
gfCNCPoint1[7593] = {X 416.6180, Y 102.7942, Z -1.3333, A 0.000, B 0.000, C 0.000 }
gfCNCPoint1[7594] = {X 417.4973, Y 102.5396, Z -1.3333, A 0.000, B 0.000, C 0.000 }
gfCNCPoint1[7595] = {X 418.3136, Y 102.1254, Z -1.3333, A 0.000, B 0.000, C 0.000 }
gfCNCPoint1[7596] = {X 419.0381, Y 101.5660, Z -1.3333, A 0.000, B 0.000, C 0.000 }
gfCNCPoint1[7597] = {X 419.6454, Y 100.8811, Z -1.3333, A 0.000, B 0.000, C 0.000 }
gfCNCPoint1[7598] = {X 420.1142, Y 100.0949, Z -1.3333, A 0.000, B 0.000, C 0.000 }
gfCNCPoint1[7599] = {X 443.7010, Y 100.0949, Z -1.3333, A 0.000, B 0.000, C 0.000 }
gfCNCPoint1[7600] = {X 443.7010, Y 90.4949, Z -1.3333, A 0.000, B 0.000, C 0.000 }
gfCNCPoint1[7601] = {X 448.3231, Y 90.4949, Z -1.3333, A 0.000, B 0.000, C 0.000 }
gfCNCPoint1[7602] = {X 448.4021, Y 90.3746, Z -1.3333, A 0.000, B 0.000, C 0.000 }
gfCNCPoint1[7603] = {X 448.4825, Y 90.2554, Z -1.3333, A 0.000, B 0.000, C 0.000 }
gfCNCPoint1[7604] = {X 445.7340, Y 89.1779, Z -1.3333, A 0.000, B 0.000, C 0.000 }
gfCNCPoint1[7605] = {X 443.7010, Y 90.4949, Z -1.3333, A 0.000, B 0.000, C 0.000 }
gfCNCPoint1[7606] = {X 443.7010, Y 92.8949, Z -1.3333, A 0.000, B 0.000, C 0.000 }
gfCNCPoint1[7607] = {X 449.7243, Y 92.8949, Z -1.3333, A 0.000, B 0.000, C 0.000 }
gfCNCPoint1[7608] = {X 450.0698, Y 92.2375, Z -1.3333, A 0.000, B 0.000, C 0.000 }
gfCNCPoint1[7609] = {X 450.4647, Y 91.6084, Z -1.3333, A 0.000, B 0.000, C 0.000 }
gfCNCPoint1[7610] = {X 451.3969, Y 90.4463, Z -1.3333, A 0.000, B 0.000, C 0.000 }
gfCNCPoint1[7611] = {X 452.4963, Y 89.4409, Z -1.3333, A 0.000, B 0.000, C 0.000 }
gfCNCPoint1[7612] = {X 452.4963, Y 89.2510, Z -1.3333, A 0.000, B 0.000, C 0.000 }
gfCNCPoint1[7613] = {X 445.4630, Y 86.4939, Z -1.3333, A 0.000, B 0.000, C 0.000 }
gfCNCPoint1[7614] = {X 435.5820, Y 92.8949, Z -1.3333, A 0.000, B 0.000, C 0.000 }
gfCNCPoint1[7615] = {X 443.7010, Y 92.8949, Z -1.3333, A 0.000, B 0.000, C 0.000 }
gfCNCPoint1[7616] = {X 443.7010, Y 95.2949, Z -1.3333, A 0.000, B 0.000, C 0.000 }
gfCNCPoint1[7617] = {X 451.3983, Y 95.2949, Z -1.3333, A 0.000, B 0.000, C 0.000 }
gfCNCPoint1[7618] = {X 451.7785, Y 94.1744, Z -1.3333, A 0.000, B 0.000, C 0.000 }
gfCNCPoint1[7619] = {X 452.3352, Y 93.1302, Z -1.3333, A 0.000, B 0.000, C 0.000 }
gfCNCPoint1[7620] = {X 453.0537, Y 92.1901, Z -1.3333, A 0.000, B 0.000, C 0.000 }
gfCNCPoint1[7621] = {X 453.9149, Y 91.3787, Z -1.3333, A 0.000, B 0.000, C 0.000 }
gfCNCPoint1[7622] = {X 454.8963, Y 90.7176, Z -1.3333, A 0.000, B 0.000, C 0.000 }
gfCNCPoint1[7623] = {X 454.8963, Y 87.6139, Z -1.3333, A 0.000, B 0.000, C 0.000 }
gfCNCPoint1[7624] = {X 445.1920, Y 83.8099, Z -1.3333, A 0.000, B 0.000, C 0.000 }
gfCNCPoint1[7625] = {X 427.4629, Y 95.2949, Z -1.3333, A 0.000, B 0.000, C 0.000 }
gfCNCPoint1[7626] = {X 443.7010, Y 95.2949, Z -1.3333, A 0.000, B 0.000, C 0.000 }
gfCNCPoint1[7627] = {X 443.7010, Y 97.6949, Z -1.3333, A 0.000, B 0.000, C 0.000 }
gfCNCPoint1[7628] = {X 453.5796, Y 97.6949, Z -1.3333, A 0.000, B 0.000, C 0.000 }
gfCNCPoint1[7629] = {X 453.5796, Y 97.0659, Z -1.3333, A 0.000, B 0.000, C 0.000 }
gfCNCPoint1[7630] = {X 453.6990, Y 95.9930, Z -1.3333, A 0.000, B 0.000, C 0.000 }
gfCNCPoint1[7631] = {X 454.0514, Y 94.9725, Z -1.3333, A 0.000, B 0.000, C 0.000 }
gfCNCPoint1[7632] = {X 454.6196, Y 94.0545, Z -1.3333, A 0.000, B 0.000, C 0.000 }
gfCNCPoint1[7633] = {X 455.3757, Y 93.2839, Z -1.3333, A 0.000, B 0.000, C 0.000 }
gfCNCPoint1[7634] = {X 456.2827, Y 92.6984, Z -1.3333, A 0.000, B 0.000, C 0.000 }
gfCNCPoint1[7635] = {X 457.2963, Y 92.3266, Z -1.3333, A 0.000, B 0.000, C 0.000 }
gfCNCPoint1[7636] = {X 457.2963, Y 85.9769, Z -1.3333, A 0.000, B 0.000, C 0.000 }
gfCNCPoint1[7637] = {X 444.9211, Y 81.1258, Z -1.3333, A 0.000, B 0.000, C 0.000 }
gfCNCPoint1[7638] = {X 420.5852, Y 96.8907, Z -1.3333, A 0.000, B 0.000, C 0.000 }
gfCNCPoint1[7639] = {X 420.5867, Y 97.0659, Z -1.3333, A 0.000, B 0.000, C 0.000 }
gfCNCPoint1[7640] = {X 420.5867, Y 97.6949, Z -1.3333, A 0.000, B 0.000, C 0.000 }
gfCNCPoint1[7641] = {X 443.7010, Y 97.6949, Z -1.3333, A 0.000, B 0.000, C 0.000 }
gfCNCPoint1[7642] = {X 443.7010, Y 100.0949, Z -1.3333, A 0.000, B 0.000, C 0.000 }
gfCNCPoint1[7643] = {X 454.0521, Y 100.0949, Z -1.3333, A 0.000, B 0.000, C 0.000 }
gfCNCPoint1[7644] = {X 454.5209, Y 100.8811, Z -1.3333, A 0.000, B 0.000, C 0.000 }
gfCNCPoint1[7645] = {X 455.1282, Y 101.5660, Z -1.3333, A 0.000, B 0.000, C 0.000 }
gfCNCPoint1[7646] = {X 455.8528, Y 102.1254, Z -1.3333, A 0.000, B 0.000, C 0.000 }
gfCNCPoint1[7647] = {X 456.6690, Y 102.5396, Z -1.3333, A 0.000, B 0.000, C 0.000 }
gfCNCPoint1[7648] = {X 457.5483, Y 102.7942, Z -1.3333, A 0.000, B 0.000, C 0.000 }
gfCNCPoint1[7649] = {X 458.4596, Y 102.8800, Z -1.3333, A 0.000, B 0.000, C 0.000 }
gfCNCPoint1[7650] = {X 475.0000, Y 102.8800, Z -1.3333, A 0.000, B 0.000, C 0.000 }
gfCNCPoint1[7651] = {X 475.9113, Y 102.7942, Z -1.3333, A 0.000, B 0.000, C 0.000 }
gfCNCPoint1[7652] = {X 476.7906, Y 102.5396, Z -1.3333, A 0.000, B 0.000, C 0.000 }
gfCNCPoint1[7653] = {X 477.6069, Y 102.1254, Z -1.3333, A 0.000, B 0.000, C 0.000 }
gfCNCPoint1[7654] = {X 478.3314, Y 101.5660, Z -1.3333, A 0.000, B 0.000, C 0.000 }
gfCNCPoint1[7655] = {X 478.9387, Y 100.8811, Z -1.3333, A 0.000, B 0.000, C 0.000 }
gfCNCPoint1[7656] = {X 479.4075, Y 100.0949, Z -1.3333, A 0.000, B 0.000, C 0.000 }
gfCNCPoint1[7657] = {X 507.6820, Y 100.0949, Z -1.3333, A 0.000, B 0.000, C 0.000 }
gfCNCPoint1[7658] = {X 507.6820, Y 107.6949, Z -1.3333, A 0.000, B 0.000, C 0.000 }
gfCNCPoint1[7659] = {X 507.6820, Y 107.6949, Z 1.6667, A 0.000, B 0.000, C 0.000 }
gfCNCPoint1[7660] = {X 507.6820, Y 107.6949, Z 11.0000, A 0.000, B 0.000, C 0.000 }
gfCNCPoint1[7661] = {X 108.5555, Y 40.9012, Z 11.0000, A 0.000, B 0.000, C 0.000 }
gfCNCPoint1[7662] = {X 108.5555, Y 40.9012, Z 2.5000, A 0.000, B 0.000, C 0.000 }
gfCNCPoint1[7663] = {X 108.5555, Y 40.9012, Z -1.3333, A 0.000, B 0.000, C 0.000 }
gfCNCPoint1[7664] = {X 108.0637, Y 42.1029, Z -1.3333, A 0.000, B 0.000, C 0.000 }
gfCNCPoint1[7665] = {X 108.0891, Y 42.0585, Z -1.3333, A 0.000, B 0.000, C 0.000 }
gfCNCPoint1[7666] = {X 108.1150, Y 42.0145, Z -1.3333, A 0.000, B 0.000, C 0.000 }
gfCNCPoint1[7667] = {X 108.5430, Y 41.3915, Z -1.3333, A 0.000, B 0.000, C 0.000 }
gfCNCPoint1[7668] = {X 109.0473, Y 40.8285, Z -1.3333, A 0.000, B 0.000, C 0.000 }
gfCNCPoint1[7669] = {X 109.0472, Y 39.6995, Z -1.3333, A 0.000, B 0.000, C 0.000 }
gfCNCPoint1[7670] = {X 108.5555, Y 40.9012, Z -1.3333, A 0.000, B 0.000, C 0.000 }
gfCNCPoint1[7671] = {X 108.5555, Y 40.9012, Z 1.6667, A 0.000, B 0.000, C 0.000 }
gfCNCPoint1[7672] = {X 108.5555, Y 40.9012, Z 11.0000, A 0.000, B 0.000, C 0.000 }
gfCNCPoint1[7673] = {X 95.6845, Y 40.8768, Z 11.0000, A 0.000, B 0.000, C 0.000 }
gfCNCPoint1[7674] = {X 95.6845, Y 40.8768, Z 2.5000, A 0.000, B 0.000, C 0.000 }
gfCNCPoint1[7675] = {X 95.6845, Y 40.8768, Z -1.3333, A 0.000, B 0.000, C 0.000 }
gfCNCPoint1[7676] = {X 95.2098, Y 39.7157, Z -1.3333, A 0.000, B 0.000, C 0.000 }
gfCNCPoint1[7677] = {X 95.2099, Y 40.8692, Z -1.3333, A 0.000, B 0.000, C 0.000 }
gfCNCPoint1[7678] = {X 95.7340, Y 41.4135, Z -1.3333, A 0.000, B 0.000, C 0.000 }
gfCNCPoint1[7679] = {X 96.1593, Y 42.0379, Z -1.3333, A 0.000, B 0.000, C 0.000 }
gfCNCPoint1[7680] = {X 95.6845, Y 40.8768, Z -1.3333, A 0.000, B 0.000, C 0.000 }
gfCNCPoint1[7681] = {X 95.6845, Y 40.8768, Z 1.6667, A 0.000, B 0.000, C 0.000 }
gfCNCPoint1[7682] = {X 95.6845, Y 40.8768, Z 11.0000, A 0.000, B 0.000, C 0.000 }
gfCNCPoint1[7683] = {X -7.6965, Y 43.1589, Z 11.0000, A 0.000, B 0.000, C 0.000 }
gfCNCPoint1[7684] = {X -7.6965, Y 43.1589, Z 1.6667, A 0.000, B 0.000, C 0.000 }
gfCNCPoint1[7685] = {X -7.6965, Y 43.1589, Z -1.3333, A 0.000, B 0.000, C 0.000 }
gfCNCPoint1[7686] = {X -3.6965, Y 30.8019, Z -1.3333, A 0.000, B 0.000, C 0.000 }
gfCNCPoint1[7687] = {X -3.3664, Y 29.8875, Z -1.3333, A 0.000, B 0.000, C 0.000 }
gfCNCPoint1[7688] = {X -2.9760, Y 28.9971, Z -1.3333, A 0.000, B 0.000, C 0.000 }
gfCNCPoint1[7689] = {X -2.3494, Y 27.8706, Z -1.3333, A 0.000, B 0.000, C 0.000 }
gfCNCPoint1[7690] = {X -1.5930, Y 26.8267, Z -1.3333, A 0.000, B 0.000, C 0.000 }
gfCNCPoint1[7691] = {X -0.7175, Y 25.8805, Z -1.3333, A 0.000, B 0.000, C 0.000 }
gfCNCPoint1[7692] = {X 0.2644, Y 25.0452, Z -1.3333, A 0.000, B 0.000, C 0.000 }
gfCNCPoint1[7693] = {X 1.3388, Y 24.3330, Z -1.3333, A 0.000, B 0.000, C 0.000 }
gfCNCPoint1[7694] = {X 0.5788, Y 23.9226, Z -1.3333, A 0.000, B 0.000, C 0.000 }
gfCNCPoint1[7695] = {X -0.0864, Y 23.3718, Z -1.3333, A 0.000, B 0.000, C 0.000 }
gfCNCPoint1[7696] = {X -0.6312, Y 22.7015, Z -1.3333, A 0.000, B 0.000, C 0.000 }
gfCNCPoint1[7697] = {X -1.0346, Y 21.9378, Z -1.3333, A 0.000, B 0.000, C 0.000 }
gfCNCPoint1[7698] = {X -3.6458, Y 15.5423, Z -1.3333, A 0.000, B 0.000, C 0.000 }
gfCNCPoint1[7699] = {X -3.6716, Y 15.4775, Z -1.3333, A 0.000, B 0.000, C 0.000 }
gfCNCPoint1[7700] = {X -3.6965, Y 15.4123, Z -1.3333, A 0.000, B 0.000, C 0.000 }
gfCNCPoint1[7701] = {X -7.6965, Y 4.6524, Z -1.3333, A 0.000, B 0.000, C 0.000 }
gfCNCPoint1[7702] = {X -7.6965, Y 4.6524, Z 1.6667, A 0.000, B 0.000, C 0.000 }
gfCNCPoint1[7703] = {X -7.6965, Y 4.6524, Z 11.0000, A 0.000, B 0.000, C 0.000 }
gfCNCPoint1[7704] = {X -7.6965, Y 16.4121, Z 11.0000, A 0.000, B 0.000, C 0.000 }
gfCNCPoint1[7705] = {X -7.6965, Y 16.4121, Z 1.6667, A 0.000, B 0.000, C 0.000 }
gfCNCPoint1[7706] = {X -7.6965, Y 16.4121, Z -1.3333, A 0.000, B 0.000, C 0.000 }
gfCNCPoint1[7707] = {X -4.8869, Y 16.4121, Z -1.3333, A 0.000, B 0.000, C 0.000 }
gfCNCPoint1[7708] = {X -3.6965, Y 12.5934, Z -1.3333, A 0.000, B 0.000, C 0.000 }
gfCNCPoint1[7709] = {X -3.6604, Y 12.4831, Z -1.3333, A 0.000, B 0.000, C 0.000 }
gfCNCPoint1[7710] = {X -3.6215, Y 12.3738, Z -1.3333, A 0.000, B 0.000, C 0.000 }
gfCNCPoint1[7711] = {X -3.1665, Y 11.4826, Z -1.3333, A 0.000, B 0.000, C 0.000 }
gfCNCPoint1[7712] = {X -2.5188, Y 10.7200, Z -1.3333, A 0.000, B 0.000, C 0.000 }
gfCNCPoint1[7713] = {X -1.7129, Y 10.1268, Z -1.3333, A 0.000, B 0.000, C 0.000 }
gfCNCPoint1[7714] = {X -1.1157, Y 9.7861, Z -1.3333, A 0.000, B 0.000, C 0.000 }
gfCNCPoint1[7715] = {X -0.2290, Y 9.4045, Z -1.3333, A 0.000, B 0.000, C 0.000 }
gfCNCPoint1[7716] = {X 0.7202, Y 9.2292, Z -1.3333, A 0.000, B 0.000, C 0.000 }
gfCNCPoint1[7717] = {X 1.6847, Y 9.2692, Z -1.3333, A 0.000, B 0.000, C 0.000 }
gfCNCPoint1[7718] = {X 2.6163, Y 9.5223, Z -1.3333, A 0.000, B 0.000, C 0.000 }
gfCNCPoint1[7719] = {X 3.3959, Y 9.1597, Z -1.3333, A 0.000, B 0.000, C 0.000 }
gfCNCPoint1[7720] = {X 4.1960, Y 8.8452, Z -1.3333, A 0.000, B 0.000, C 0.000 }
gfCNCPoint1[7721] = {X 6.1070, Y 8.1764, Z -1.3333, A 0.000, B 0.000, C 0.000 }
gfCNCPoint1[7722] = {X 8.0685, Y 7.6749, Z -1.3333, A 0.000, B 0.000, C 0.000 }
gfCNCPoint1[7723] = {X 10.0659, Y 7.3444, Z -1.3333, A 0.000, B 0.000, C 0.000 }
gfCNCPoint1[7724] = {X 12.0844, Y 7.1873, Z -1.3333, A 0.000, B 0.000, C 0.000 }
gfCNCPoint1[7725] = {X 14.1089, Y 7.2048, Z -1.3333, A 0.000, B 0.000, C 0.000 }
gfCNCPoint1[7726] = {X 16.1243, Y 7.3968, Z -1.3333, A 0.000, B 0.000, C 0.000 }
gfCNCPoint1[7727] = {X 17.9475, Y 7.7305, Z -1.3333, A 0.000, B 0.000, C 0.000 }
gfCNCPoint1[7728] = {X 19.7250, Y 8.2556, Z -1.3333, A 0.000, B 0.000, C 0.000 }
gfCNCPoint1[7729] = {X 21.4369, Y 8.9662, Z -1.3333, A 0.000, B 0.000, C 0.000 }
gfCNCPoint1[7730] = {X 23.0637, Y 9.8542, Z -1.3333, A 0.000, B 0.000, C 0.000 }
gfCNCPoint1[7731] = {X 24.5873, Y 10.9096, Z -1.3333, A 0.000, B 0.000, C 0.000 }
gfCNCPoint1[7732] = {X 25.6720, Y 11.8588, Z -1.3333, A 0.000, B 0.000, C 0.000 }
gfCNCPoint1[7733] = {X 26.6451, Y 12.9220, Z -1.3333, A 0.000, B 0.000, C 0.000 }
gfCNCPoint1[7734] = {X 27.4946, Y 14.0863, Z -1.3333, A 0.000, B 0.000, C 0.000 }
gfCNCPoint1[7735] = {X 28.2102, Y 15.3374, Z -1.3333, A 0.000, B 0.000, C 0.000 }
gfCNCPoint1[7736] = {X 28.7831, Y 16.6600, Z -1.3333, A 0.000, B 0.000, C 0.000 }
gfCNCPoint1[7737] = {X 29.2572, Y 18.3163, Z -1.3333, A 0.000, B 0.000, C 0.000 }
gfCNCPoint1[7738] = {X 29.5386, Y 20.0161, Z -1.3333, A 0.000, B 0.000, C 0.000 }
gfCNCPoint1[7739] = {X 29.6235, Y 21.7368, Z -1.3333, A 0.000, B 0.000, C 0.000 }
gfCNCPoint1[7740] = {X 29.5110, Y 23.4560, Z -1.3333, A 0.000, B 0.000, C 0.000 }
gfCNCPoint1[7741] = {X 29.2023, Y 25.1510, Z -1.3333, A 0.000, B 0.000, C 0.000 }
gfCNCPoint1[7742] = {X 28.7603, Y 26.5972, Z -1.3333, A 0.000, B 0.000, C 0.000 }
gfCNCPoint1[7743] = {X 28.1353, Y 27.9742, Z -1.3333, A 0.000, B 0.000, C 0.000 }
gfCNCPoint1[7744] = {X 27.3377, Y 29.2589, Z -1.3333, A 0.000, B 0.000, C 0.000 }
gfCNCPoint1[7745] = {X 26.3808, Y 30.4299, Z -1.3333, A 0.000, B 0.000, C 0.000 }
gfCNCPoint1[7746] = {X 25.2808, Y 31.4675, Z -1.3333, A 0.000, B 0.000, C 0.000 }
gfCNCPoint1[7747] = {X 26.0849, Y 31.8096, Z -1.3333, A 0.000, B 0.000, C 0.000 }
gfCNCPoint1[7748] = {X 26.8038, Y 32.3066, Z -1.3333, A 0.000, B 0.000, C 0.000 }
gfCNCPoint1[7749] = {X 27.4079, Y 32.9380, Z -1.3333, A 0.000, B 0.000, C 0.000 }
gfCNCPoint1[7750] = {X 27.8726, Y 33.6781, Z -1.3333, A 0.000, B 0.000, C 0.000 }
gfCNCPoint1[7751] = {X 30.9100, Y 39.9530, Z -1.3333, A 0.000, B 0.000, C 0.000 }
gfCNCPoint1[7752] = {X 31.2306, Y 40.8622, Z -1.3333, A 0.000, B 0.000, C 0.000 }
gfCNCPoint1[7753] = {X 31.3415, Y 41.8197, Z -1.3333, A 0.000, B 0.000, C 0.000 }
gfCNCPoint1[7754] = {X 31.2374, Y 42.7781, Z -1.3333, A 0.000, B 0.000, C 0.000 }
gfCNCPoint1[7755] = {X 30.9234, Y 43.6895, Z -1.3333, A 0.000, B 0.000, C 0.000 }
gfCNCPoint1[7756] = {X 30.4150, Y 44.5085, Z -1.3333, A 0.000, B 0.000, C 0.000 }
gfCNCPoint1[7757] = {X 29.7377, Y 45.1945, Z -1.3333, A 0.000, B 0.000, C 0.000 }
gfCNCPoint1[7758] = {X 29.2013, Y 45.6282, Z -1.3333, A 0.000, B 0.000, C 0.000 }
gfCNCPoint1[7759] = {X 28.4963, Y 46.0911, Z -1.3333, A 0.000, B 0.000, C 0.000 }
gfCNCPoint1[7760] = {X 27.7151, Y 46.4089, Z -1.3333, A 0.000, B 0.000, C 0.000 }
gfCNCPoint1[7761] = {X 26.8872, Y 46.5696, Z -1.3333, A 0.000, B 0.000, C 0.000 }
gfCNCPoint1[7762] = {X 26.0438, Y 46.5671, Z -1.3333, A 0.000, B 0.000, C 0.000 }
gfCNCPoint1[7763] = {X 25.2169, Y 46.4014, Z -1.3333, A 0.000, B 0.000, C 0.000 }
gfCNCPoint1[7764] = {X 23.1982, Y 47.4600, Z -1.3333, A 0.000, B 0.000, C 0.000 }
gfCNCPoint1[7765] = {X 21.1011, Y 48.3534, Z -1.3333, A 0.000, B 0.000, C 0.000 }
gfCNCPoint1[7766] = {X 18.9393, Y 49.0761, Z -1.3333, A 0.000, B 0.000, C 0.000 }
gfCNCPoint1[7767] = {X 18.4459, Y 49.2128, Z -1.3333, A 0.000, B 0.000, C 0.000 }
gfCNCPoint1[7768] = {X 16.5824, Y 49.6439, Z -1.3333, A 0.000, B 0.000, C 0.000 }
gfCNCPoint1[7769] = {X 14.6888, Y 49.9134, Z -1.3333, A 0.000, B 0.000, C 0.000 }
gfCNCPoint1[7770] = {X 12.7790, Y 50.0195, Z -1.3333, A 0.000, B 0.000, C 0.000 }
gfCNCPoint1[7771] = {X 10.8672, Y 49.9612, Z -1.3333, A 0.000, B 0.000, C 0.000 }
gfCNCPoint1[7772] = {X 8.9675, Y 49.7390, Z -1.3333, A 0.000, B 0.000, C 0.000 }
gfCNCPoint1[7773] = {X 7.3410, Y 49.4309, Z -1.3333, A 0.000, B 0.000, C 0.000 }
gfCNCPoint1[7774] = {X 5.7518, Y 48.9671, Z -1.3333, A 0.000, B 0.000, C 0.000 }
gfCNCPoint1[7775] = {X 4.2147, Y 48.3522, Z -1.3333, A 0.000, B 0.000, C 0.000 }
gfCNCPoint1[7776] = {X 2.7442, Y 47.5918, Z -1.3333, A 0.000, B 0.000, C 0.000 }
gfCNCPoint1[7777] = {X 1.3540, Y 46.6930, Z -1.3333, A 0.000, B 0.000, C 0.000 }
gfCNCPoint1[7778] = {X 0.0286, Y 45.6272, Z -1.3333, A 0.000, B 0.000, C 0.000 }
gfCNCPoint1[7779] = {X -1.1495, Y 44.4005, Z -1.3333, A 0.000, B 0.000, C 0.000 }
gfCNCPoint1[7780] = {X -2.1609, Y 43.0332, Z -1.3333, A 0.000, B 0.000, C 0.000 }
gfCNCPoint1[7781] = {X -2.9891, Y 41.5477, Z -1.3333, A 0.000, B 0.000, C 0.000 }
gfCNCPoint1[7782] = {X -3.6204, Y 39.9684, Z -1.3333, A 0.000, B 0.000, C 0.000 }
gfCNCPoint1[7783] = {X -3.6590, Y 39.8485, Z -1.3333, A 0.000, B 0.000, C 0.000 }
gfCNCPoint1[7784] = {X -3.6965, Y 39.7283, Z -1.3333, A 0.000, B 0.000, C 0.000 }
gfCNCPoint1[7785] = {X -4.8676, Y 35.9036, Z -1.3333, A 0.000, B 0.000, C 0.000 }
gfCNCPoint1[7786] = {X -7.9895, Y 36.0311, Z -1.3333, A 0.000, B 0.000, C 0.000 }
gfCNCPoint1[7787] = {X -7.9895, Y 36.0311, Z 1.6667, A 0.000, B 0.000, C 0.000 }
gfCNCPoint1[7788] = {X -7.9895, Y 36.0311, Z 11.0000, A 0.000, B 0.000, C 0.000 }
gfCNCPoint1[7789] = {X 608.0000, Y 40.1206, Z 11.0000, A 0.000, B 0.000, C 0.000 }
gfCNCPoint1[7790] = {X 608.0000, Y 40.1206, Z 1.6667, A 0.000, B 0.000, C 0.000 }
gfCNCPoint1[7791] = {X 608.0000, Y 40.1206, Z -1.3333, A 0.000, B 0.000, C 0.000 }
gfCNCPoint1[7792] = {X 603.6965, Y 47.2358, Z -1.3333, A 0.000, B 0.000, C 0.000 }
gfCNCPoint1[7793] = {X 603.6632, Y 47.2898, Z -1.3333, A 0.000, B 0.000, C 0.000 }
gfCNCPoint1[7794] = {X 603.6292, Y 47.3433, Z -1.3333, A 0.000, B 0.000, C 0.000 }
gfCNCPoint1[7795] = {X 603.0929, Y 48.0160, Z -1.3333, A 0.000, B 0.000, C 0.000 }
gfCNCPoint1[7796] = {X 602.4338, Y 48.5691, Z -1.3333, A 0.000, B 0.000, C 0.000 }
gfCNCPoint1[7797] = {X 601.6783, Y 48.9807, Z -1.3333, A 0.000, B 0.000, C 0.000 }
gfCNCPoint1[7798] = {X 600.8561, Y 49.2343, Z -1.3333, A 0.000, B 0.000, C 0.000 }
gfCNCPoint1[7799] = {X 600.0000, Y 49.3200, Z -1.3333, A 0.000, B 0.000, C 0.000 }
gfCNCPoint1[7800] = {X 593.5565, Y 49.3200, Z -1.3333, A 0.000, B 0.000, C 0.000 }
gfCNCPoint1[7801] = {X 592.5952, Y 49.2117, Z -1.3333, A 0.000, B 0.000, C 0.000 }
gfCNCPoint1[7802] = {X 591.6822, Y 48.8922, Z -1.3333, A 0.000, B 0.000, C 0.000 }
gfCNCPoint1[7803] = {X 590.8631, Y 48.3775, Z -1.3333, A 0.000, B 0.000, C 0.000 }
gfCNCPoint1[7804] = {X 590.1790, Y 47.6935, Z -1.3333, A 0.000, B 0.000, C 0.000 }
gfCNCPoint1[7805] = {X 589.6643, Y 46.8744, Z -1.3333, A 0.000, B 0.000, C 0.000 }
gfCNCPoint1[7806] = {X 589.3448, Y 45.9613, Z -1.3333, A 0.000, B 0.000, C 0.000 }
gfCNCPoint1[7807] = {X 589.2365, Y 45.0000, Z -1.3333, A 0.000, B 0.000, C 0.000 }
gfCNCPoint1[7808] = {X 589.2365, Y 44.0643, Z -1.3333, A 0.000, B 0.000, C 0.000 }
gfCNCPoint1[7809] = {X 589.3416, Y 43.1363, Z -1.3333, A 0.000, B 0.000, C 0.000 }
gfCNCPoint1[7810] = {X 589.6416, Y 42.2518, Z -1.3333, A 0.000, B 0.000, C 0.000 }
gfCNCPoint1[7811] = {X 590.1229, Y 41.4515, Z -1.3333, A 0.000, B 0.000, C 0.000 }
gfCNCPoint1[7812] = {X 590.7634, Y 40.7718, Z -1.3333, A 0.000, B 0.000, C 0.000 }
gfCNCPoint1[7813] = {X 590.7637, Y 33.5287, Z -1.3333, A 0.000, B 0.000, C 0.000 }
gfCNCPoint1[7814] = {X 585.4453, Y 46.6524, Z -1.3333, A 0.000, B 0.000, C 0.000 }
gfCNCPoint1[7815] = {X 585.0755, Y 47.3550, Z -1.3333, A 0.000, B 0.000, C 0.000 }
gfCNCPoint1[7816] = {X 584.5834, Y 47.9780, Z -1.3333, A 0.000, B 0.000, C 0.000 }
gfCNCPoint1[7817] = {X 583.9856, Y 48.5004, Z -1.3333, A 0.000, B 0.000, C 0.000 }
gfCNCPoint1[7818] = {X 583.3023, Y 48.9046, Z -1.3333, A 0.000, B 0.000, C 0.000 }
gfCNCPoint1[7819] = {X 582.3585, Y 49.2242, Z -1.3333, A 0.000, B 0.000, C 0.000 }
gfCNCPoint1[7820] = {X 581.3666, Y 49.3191, Z -1.3333, A 0.000, B 0.000, C 0.000 }
gfCNCPoint1[7821] = {X 580.3794, Y 49.1842, Z -1.3333, A 0.000, B 0.000, C 0.000 }
gfCNCPoint1[7822] = {X 579.4493, Y 48.8268, Z -1.3333, A 0.000, B 0.000, C 0.000 }
gfCNCPoint1[7823] = {X 578.6259, Y 48.2657, Z -1.3333, A 0.000, B 0.000, C 0.000 }
gfCNCPoint1[7824] = {X 577.9529, Y 47.5309, Z -1.3333, A 0.000, B 0.000, C 0.000 }
gfCNCPoint1[7825] = {X 577.4662, Y 46.6615, Z -1.3333, A 0.000, B 0.000, C 0.000 }
gfCNCPoint1[7826] = {X 572.0176, Y 33.3383, Z -1.3333, A 0.000, B 0.000, C 0.000 }
gfCNCPoint1[7827] = {X 572.0180, Y 40.7702, Z -1.3333, A 0.000, B 0.000, C 0.000 }
gfCNCPoint1[7828] = {X 572.6567, Y 41.4411, Z -1.3333, A 0.000, B 0.000, C 0.000 }
gfCNCPoint1[7829] = {X 573.1376, Y 42.2327, Z -1.3333, A 0.000, B 0.000, C 0.000 }
gfCNCPoint1[7830] = {X 573.4388, Y 43.1087, Z -1.3333, A 0.000, B 0.000, C 0.000 }
gfCNCPoint1[7831] = {X 573.5463, Y 44.0287, Z -1.3333, A 0.000, B 0.000, C 0.000 }
gfCNCPoint1[7832] = {X 573.5464, Y 45.0000, Z -1.3333, A 0.000, B 0.000, C 0.000 }
gfCNCPoint1[7833] = {X 573.4381, Y 45.9613, Z -1.3333, A 0.000, B 0.000, C 0.000 }
gfCNCPoint1[7834] = {X 573.1186, Y 46.8744, Z -1.3333, A 0.000, B 0.000, C 0.000 }
gfCNCPoint1[7835] = {X 572.6039, Y 47.6935, Z -1.3333, A 0.000, B 0.000, C 0.000 }
gfCNCPoint1[7836] = {X 571.9199, Y 48.3775, Z -1.3333, A 0.000, B 0.000, C 0.000 }
gfCNCPoint1[7837] = {X 571.1008, Y 48.8922, Z -1.3333, A 0.000, B 0.000, C 0.000 }
gfCNCPoint1[7838] = {X 570.1877, Y 49.2117, Z -1.3333, A 0.000, B 0.000, C 0.000 }
gfCNCPoint1[7839] = {X 569.2264, Y 49.3200, Z -1.3333, A 0.000, B 0.000, C 0.000 }
gfCNCPoint1[7840] = {X 562.4443, Y 49.3200, Z -1.3333, A 0.000, B 0.000, C 0.000 }
gfCNCPoint1[7841] = {X 561.4830, Y 49.2117, Z -1.3333, A 0.000, B 0.000, C 0.000 }
gfCNCPoint1[7842] = {X 560.5699, Y 48.8922, Z -1.3333, A 0.000, B 0.000, C 0.000 }
gfCNCPoint1[7843] = {X 559.7508, Y 48.3775, Z -1.3333, A 0.000, B 0.000, C 0.000 }
gfCNCPoint1[7844] = {X 559.0668, Y 47.6935, Z -1.3333, A 0.000, B 0.000, C 0.000 }
gfCNCPoint1[7845] = {X 558.5521, Y 46.8744, Z -1.3333, A 0.000, B 0.000, C 0.000 }
gfCNCPoint1[7846] = {X 558.2326, Y 45.9613, Z -1.3333, A 0.000, B 0.000, C 0.000 }
gfCNCPoint1[7847] = {X 558.1243, Y 45.0000, Z -1.3333, A 0.000, B 0.000, C 0.000 }
gfCNCPoint1[7848] = {X 558.1243, Y 44.0644, Z -1.3333, A 0.000, B 0.000, C 0.000 }
gfCNCPoint1[7849] = {X 558.2292, Y 43.1360, Z -1.3333, A 0.000, B 0.000, C 0.000 }
gfCNCPoint1[7850] = {X 558.5295, Y 42.2512, Z -1.3333, A 0.000, B 0.000, C 0.000 }
gfCNCPoint1[7851] = {X 559.0115, Y 41.4508, Z -1.3333, A 0.000, B 0.000, C 0.000 }
gfCNCPoint1[7852] = {X 559.6530, Y 40.7715, Z -1.3333, A 0.000, B 0.000, C 0.000 }
gfCNCPoint1[7853] = {X 559.6530, Y 9.2312, Z -1.3333, A 0.000, B 0.000, C 0.000 }
gfCNCPoint1[7854] = {X 559.0141, Y 8.5601, Z -1.3333, A 0.000, B 0.000, C 0.000 }
gfCNCPoint1[7855] = {X 558.5330, Y 7.7683, Z -1.3333, A 0.000, B 0.000, C 0.000 }
gfCNCPoint1[7856] = {X 558.2319, Y 6.8921, Z -1.3333, A 0.000, B 0.000, C 0.000 }
gfCNCPoint1[7857] = {X 558.1245, Y 5.9718, Z -1.3333, A 0.000, B 0.000, C 0.000 }
gfCNCPoint1[7858] = {X 558.1243, Y 5.0000, Z -1.3333, A 0.000, B 0.000, C 0.000 }
gfCNCPoint1[7859] = {X 558.2326, Y 4.0387, Z -1.3333, A 0.000, B 0.000, C 0.000 }
gfCNCPoint1[7860] = {X 558.5521, Y 3.1256, Z -1.3333, A 0.000, B 0.000, C 0.000 }
gfCNCPoint1[7861] = {X 559.0668, Y 2.3065, Z -1.3333, A 0.000, B 0.000, C 0.000 }
gfCNCPoint1[7862] = {X 559.7508, Y 1.6225, Z -1.3333, A 0.000, B 0.000, C 0.000 }
gfCNCPoint1[7863] = {X 560.5699, Y 1.1078, Z -1.3333, A 0.000, B 0.000, C 0.000 }
gfCNCPoint1[7864] = {X 561.4830, Y 0.7883, Z -1.3333, A 0.000, B 0.000, C 0.000 }
gfCNCPoint1[7865] = {X 562.4443, Y 0.6800, Z -1.3333, A 0.000, B 0.000, C 0.000 }
gfCNCPoint1[7866] = {X 570.9376, Y 0.6800, Z -1.3333, A 0.000, B 0.000, C 0.000 }
gfCNCPoint1[7867] = {X 571.8988, Y 0.7883, Z -1.3333, A 0.000, B 0.000, C 0.000 }
gfCNCPoint1[7868] = {X 572.8119, Y 1.1078, Z -1.3333, A 0.000, B 0.000, C 0.000 }
gfCNCPoint1[7869] = {X 573.6310, Y 1.6225, Z -1.3333, A 0.000, B 0.000, C 0.000 }
gfCNCPoint1[7870] = {X 574.3151, Y 2.3065, Z -1.3333, A 0.000, B 0.000, C 0.000 }
gfCNCPoint1[7871] = {X 574.8297, Y 3.1256, Z -1.3333, A 0.000, B 0.000, C 0.000 }
gfCNCPoint1[7872] = {X 575.1492, Y 4.0387, Z -1.3333, A 0.000, B 0.000, C 0.000 }
gfCNCPoint1[7873] = {X 575.2576, Y 5.0000, Z -1.3333, A 0.000, B 0.000, C 0.000 }
gfCNCPoint1[7874] = {X 575.2576, Y 5.9342, Z -1.3333, A 0.000, B 0.000, C 0.000 }
gfCNCPoint1[7875] = {X 575.1834, Y 6.7310, Z -1.3333, A 0.000, B 0.000, C 0.000 }
gfCNCPoint1[7876] = {X 574.9636, Y 7.5005, Z -1.3333, A 0.000, B 0.000, C 0.000 }
gfCNCPoint1[7877] = {X 574.6056, Y 8.2162, Z -1.3333, A 0.000, B 0.000, C 0.000 }
gfCNCPoint1[7878] = {X 581.1909, Y 24.3712, Z -1.3333, A 0.000, B 0.000, C 0.000 }
gfCNCPoint1[7879] = {X 587.8461, Y 8.0947, Z -1.3333, A 0.000, B 0.000, C 0.000 }
gfCNCPoint1[7880] = {X 587.5318, Y 7.4234, Z -1.3333, A 0.000, B 0.000, C 0.000 }
gfCNCPoint1[7881] = {X 587.3369, Y 6.7084, Z -1.3333, A 0.000, B 0.000, C 0.000 }
gfCNCPoint1[7882] = {X 587.2671, Y 5.9705, Z -1.3333, A 0.000, B 0.000, C 0.000 }
gfCNCPoint1[7883] = {X 587.2670, Y 5.0000, Z -1.3333, A 0.000, B 0.000, C 0.000 }
gfCNCPoint1[7884] = {X 587.3753, Y 4.0387, Z -1.3333, A 0.000, B 0.000, C 0.000 }
gfCNCPoint1[7885] = {X 587.6948, Y 3.1256, Z -1.3333, A 0.000, B 0.000, C 0.000 }
gfCNCPoint1[7886] = {X 588.2094, Y 2.3065, Z -1.3333, A 0.000, B 0.000, C 0.000 }
gfCNCPoint1[7887] = {X 588.8935, Y 1.6225, Z -1.3333, A 0.000, B 0.000, C 0.000 }
gfCNCPoint1[7888] = {X 589.7126, Y 1.1078, Z -1.3333, A 0.000, B 0.000, C 0.000 }
gfCNCPoint1[7889] = {X 590.6257, Y 0.7883, Z -1.3333, A 0.000, B 0.000, C 0.000 }
gfCNCPoint1[7890] = {X 591.5870, Y 0.6800, Z -1.3333, A 0.000, B 0.000, C 0.000 }
gfCNCPoint1[7891] = {X 600.0000, Y 0.6800, Z -1.3333, A 0.000, B 0.000, C 0.000 }
gfCNCPoint1[7892] = {X 600.8561, Y 0.7657, Z -1.3333, A 0.000, B 0.000, C 0.000 }
gfCNCPoint1[7893] = {X 601.6783, Y 1.0193, Z -1.3333, A 0.000, B 0.000, C 0.000 }
gfCNCPoint1[7894] = {X 602.4338, Y 1.4309, Z -1.3333, A 0.000, B 0.000, C 0.000 }
gfCNCPoint1[7895] = {X 603.0929, Y 1.9840, Z -1.3333, A 0.000, B 0.000, C 0.000 }
gfCNCPoint1[7896] = {X 603.6292, Y 2.6567, Z -1.3333, A 0.000, B 0.000, C 0.000 }
gfCNCPoint1[7897] = {X 603.6632, Y 2.7102, Z -1.3333, A 0.000, B 0.000, C 0.000 }
gfCNCPoint1[7898] = {X 603.6965, Y 2.7642, Z -1.3333, A 0.000, B 0.000, C 0.000 }
gfCNCPoint1[7899] = {X 608.0000, Y 9.8794, Z -1.3333, A 0.000, B 0.000, C 0.000 }
gfCNCPoint1[7900] = {X 608.0000, Y 9.8794, Z 1.6667, A 0.000, B 0.000, C 0.000 }
gfCNCPoint1[7901] = {X 608.0000, Y 9.8794, Z 11.0000, A 0.000, B 0.000, C 0.000 }
gfCNCPoint1[7902] = {X -7.6965, Y 16.7859, Z 11.0000, A 0.000, B 0.000, C 0.000 }
gfCNCPoint1[7903] = {X -7.6965, Y 16.7859, Z 1.6667, A 0.000, B 0.000, C 0.000 }
gfCNCPoint1[7904] = {X -7.6965, Y 16.7859, Z -1.3333, A 0.000, B 0.000, C 0.000 }
gfCNCPoint1[7905] = {X -4.6248, Y 16.7859, Z -1.3333, A 0.000, B 0.000, C 0.000 }
gfCNCPoint1[7906] = {X -3.6965, Y 12.8951, Z -1.3333, A 0.000, B 0.000, C 0.000 }
gfCNCPoint1[7907] = {X -3.6290, Y 12.6461, Z -1.3333, A 0.000, B 0.000, C 0.000 }
gfCNCPoint1[7908] = {X -3.5465, Y 12.4017, Z -1.3333, A 0.000, B 0.000, C 0.000 }
gfCNCPoint1[7909] = {X -3.1000, Y 11.5270, Z -1.3333, A 0.000, B 0.000, C 0.000 }
gfCNCPoint1[7910] = {X -2.4642, Y 10.7785, Z -1.3333, A 0.000, B 0.000, C 0.000 }
gfCNCPoint1[7911] = {X -1.6733, Y 10.1963, Z -1.3333, A 0.000, B 0.000, C 0.000 }
gfCNCPoint1[7912] = {X -1.0761, Y 9.8556, Z -1.3333, A 0.000, B 0.000, C 0.000 }
gfCNCPoint1[7913] = {X -0.1973, Y 9.4784, Z -1.3333, A 0.000, B 0.000, C 0.000 }
gfCNCPoint1[7914] = {X 0.7437, Y 9.3078, Z -1.3333, A 0.000, B 0.000, C 0.000 }
gfCNCPoint1[7915] = {X 1.6990, Y 9.3524, Z -1.3333, A 0.000, B 0.000, C 0.000 }
gfCNCPoint1[7916] = {X 2.6200, Y 9.6100, Z -1.3333, A 0.000, B 0.000, C 0.000 }
gfCNCPoint1[7917] = {X 3.4115, Y 9.2401, Z -1.3333, A 0.000, B 0.000, C 0.000 }
gfCNCPoint1[7918] = {X 4.2244, Y 8.9200, Z -1.3333, A 0.000, B 0.000, C 0.000 }
gfCNCPoint1[7919] = {X 6.1290, Y 8.2533, Z -1.3333, A 0.000, B 0.000, C 0.000 }
gfCNCPoint1[7920] = {X 8.0841, Y 7.7534, Z -1.3333, A 0.000, B 0.000, C 0.000 }
gfCNCPoint1[7921] = {X 10.0750, Y 7.4238, Z -1.3333, A 0.000, B 0.000, C 0.000 }
gfCNCPoint1[7922] = {X 12.0869, Y 7.2672, Z -1.3333, A 0.000, B 0.000, C 0.000 }
gfCNCPoint1[7923] = {X 14.1048, Y 7.2847, Z -1.3333, A 0.000, B 0.000, C 0.000 }
gfCNCPoint1[7924] = {X 16.1137, Y 7.4761, Z -1.3333, A 0.000, B 0.000, C 0.000 }
gfCNCPoint1[7925] = {X 17.9286, Y 7.8082, Z -1.3333, A 0.000, B 0.000, C 0.000 }
gfCNCPoint1[7926] = {X 19.6981, Y 8.3309, Z -1.3333, A 0.000, B 0.000, C 0.000 }
gfCNCPoint1[7927] = {X 21.4022, Y 9.0383, Z -1.3333, A 0.000, B 0.000, C 0.000 }
gfCNCPoint1[7928] = {X 23.0217, Y 9.9222, Z -1.3333, A 0.000, B 0.000, C 0.000 }
gfCNCPoint1[7929] = {X 24.5383, Y 10.9729, Z -1.3333, A 0.000, B 0.000, C 0.000 }
gfCNCPoint1[7930] = {X 25.6163, Y 11.9162, Z -1.3333, A 0.000, B 0.000, C 0.000 }
gfCNCPoint1[7931] = {X 26.5833, Y 12.9728, Z -1.3333, A 0.000, B 0.000, C 0.000 }
gfCNCPoint1[7932] = {X 27.4276, Y 14.1299, Z -1.3333, A 0.000, B 0.000, C 0.000 }
gfCNCPoint1[7933] = {X 28.1387, Y 15.3733, Z -1.3333, A 0.000, B 0.000, C 0.000 }
gfCNCPoint1[7934] = {X 28.7080, Y 16.6876, Z -1.3333, A 0.000, B 0.000, C 0.000 }
gfCNCPoint1[7935] = {X 29.1794, Y 18.3350, Z -1.3333, A 0.000, B 0.000, C 0.000 }
gfCNCPoint1[7936] = {X 29.4591, Y 20.0255, Z -1.3333, A 0.000, B 0.000, C 0.000 }
gfCNCPoint1[7937] = {X 29.5435, Y 21.7368, Z -1.3333, A 0.000, B 0.000, C 0.000 }
gfCNCPoint1[7938] = {X 29.4315, Y 23.4466, Z -1.3333, A 0.000, B 0.000, C 0.000 }
gfCNCPoint1[7939] = {X 29.1245, Y 25.1324, Z -1.3333, A 0.000, B 0.000, C 0.000 }
gfCNCPoint1[7940] = {X 28.6748, Y 26.5971, Z -1.3333, A 0.000, B 0.000, C 0.000 }
gfCNCPoint1[7941] = {X 28.0361, Y 27.9897, Z -1.3333, A 0.000, B 0.000, C 0.000 }
gfCNCPoint1[7942] = {X 27.2195, Y 29.2861, Z -1.3333, A 0.000, B 0.000, C 0.000 }
gfCNCPoint1[7943] = {X 26.2392, Y 30.4637, Z -1.3333, A 0.000, B 0.000, C 0.000 }
gfCNCPoint1[7944] = {X 25.1123, Y 31.5018, Z -1.3333, A 0.000, B 0.000, C 0.000 }
gfCNCPoint1[7945] = {X 25.2519, Y 31.5423, Z -1.3333, A 0.000, B 0.000, C 0.000 }
gfCNCPoint1[7946] = {X 25.3900, Y 31.5876, Z -1.3333, A 0.000, B 0.000, C 0.000 }
gfCNCPoint1[7947] = {X 26.1376, Y 31.9315, Z -1.3333, A 0.000, B 0.000, C 0.000 }
gfCNCPoint1[7948] = {X 26.8047, Y 32.4133, Z -1.3333, A 0.000, B 0.000, C 0.000 }
gfCNCPoint1[7949] = {X 27.3662, Y 33.0149, Z -1.3333, A 0.000, B 0.000, C 0.000 }
gfCNCPoint1[7950] = {X 27.8009, Y 33.7136, Z -1.3333, A 0.000, B 0.000, C 0.000 }
gfCNCPoint1[7951] = {X 30.8380, Y 39.9879, Z -1.3333, A 0.000, B 0.000, C 0.000 }
gfCNCPoint1[7952] = {X 31.1526, Y 40.8802, Z -1.3333, A 0.000, B 0.000, C 0.000 }
gfCNCPoint1[7953] = {X 31.2615, Y 41.8200, Z -1.3333, A 0.000, B 0.000, C 0.000 }
gfCNCPoint1[7954] = {X 31.1593, Y 42.7606, Z -1.3333, A 0.000, B 0.000, C 0.000 }
gfCNCPoint1[7955] = {X 30.8511, Y 43.6551, Z -1.3333, A 0.000, B 0.000, C 0.000 }
gfCNCPoint1[7956] = {X 30.3522, Y 44.4590, Z -1.3333, A 0.000, B 0.000, C 0.000 }
gfCNCPoint1[7957] = {X 29.6874, Y 45.1323, Z -1.3333, A 0.000, B 0.000, C 0.000 }
gfCNCPoint1[7958] = {X 29.1511, Y 45.5659, Z -1.3333, A 0.000, B 0.000, C 0.000 }
gfCNCPoint1[7959] = {X 28.4530, Y 46.0235, Z -1.3333, A 0.000, B 0.000, C 0.000 }
gfCNCPoint1[7960] = {X 27.6791, Y 46.3361, Z -1.3333, A 0.000, B 0.000, C 0.000 }
gfCNCPoint1[7961] = {X 26.8590, Y 46.4918, Z -1.3333, A 0.000, B 0.000, C 0.000 }
gfCNCPoint1[7962] = {X 26.0243, Y 46.4846, Z -1.3333, A 0.000, B 0.000, C 0.000 }
gfCNCPoint1[7963] = {X 25.2071, Y 46.3147, Z -1.3333, A 0.000, B 0.000, C 0.000 }
gfCNCPoint1[7964] = {X 23.1849, Y 47.3777, Z -1.3333, A 0.000, B 0.000, C 0.000 }
gfCNCPoint1[7965] = {X 21.0836, Y 48.2745, Z -1.3333, A 0.000, B 0.000, C 0.000 }
gfCNCPoint1[7966] = {X 18.9170, Y 48.9992, Z -1.3333, A 0.000, B 0.000, C 0.000 }
gfCNCPoint1[7967] = {X 18.4245, Y 49.1357, Z -1.3333, A 0.000, B 0.000, C 0.000 }
gfCNCPoint1[7968] = {X 16.5676, Y 49.5653, Z -1.3333, A 0.000, B 0.000, C 0.000 }
gfCNCPoint1[7969] = {X 14.6806, Y 49.8339, Z -1.3333, A 0.000, B 0.000, C 0.000 }
gfCNCPoint1[7970] = {X 12.7776, Y 49.9395, Z -1.3333, A 0.000, B 0.000, C 0.000 }
gfCNCPoint1[7971] = {X 10.8725, Y 49.8814, Z -1.3333, A 0.000, B 0.000, C 0.000 }
gfCNCPoint1[7972] = {X 8.9794, Y 49.6599, Z -1.3333, A 0.000, B 0.000, C 0.000 }
gfCNCPoint1[7973] = {X 7.3602, Y 49.3532, Z -1.3333, A 0.000, B 0.000, C 0.000 }
gfCNCPoint1[7974] = {X 5.7782, Y 48.8916, Z -1.3333, A 0.000, B 0.000, C 0.000 }
gfCNCPoint1[7975] = {X 4.2481, Y 48.2795, Z -1.3333, A 0.000, B 0.000, C 0.000 }
gfCNCPoint1[7976] = {X 2.7843, Y 47.5225, Z -1.3333, A 0.000, B 0.000, C 0.000 }
gfCNCPoint1[7977] = {X 1.4004, Y 46.6278, Z -1.3333, A 0.000, B 0.000, C 0.000 }
gfCNCPoint1[7978] = {X 0.0829, Y 45.5684, Z -1.3333, A 0.000, B 0.000, C 0.000 }
gfCNCPoint1[7979] = {X -1.0882, Y 44.3491, Z -1.3333, A 0.000, B 0.000, C 0.000 }
gfCNCPoint1[7980] = {X -2.0936, Y 42.9900, Z -1.3333, A 0.000, B 0.000, C 0.000 }
gfCNCPoint1[7981] = {X -2.9169, Y 41.5134, Z -1.3333, A 0.000, B 0.000, C 0.000 }
gfCNCPoint1[7982] = {X -3.5444, Y 39.9436, Z -1.3333, A 0.000, B 0.000, C 0.000 }
gfCNCPoint1[7983] = {X -3.6229, Y 39.6953, Z -1.3333, A 0.000, B 0.000, C 0.000 }
gfCNCPoint1[7984] = {X -3.6965, Y 39.4456, Z -1.3333, A 0.000, B 0.000, C 0.000 }
gfCNCPoint1[7985] = {X -4.7889, Y 35.5976, Z -1.3333, A 0.000, B 0.000, C 0.000 }
gfCNCPoint1[7986] = {X -8.0008, Y 35.6638, Z -1.3333, A 0.000, B 0.000, C 0.000 }
gfCNCPoint1[7987] = {X -8.0008, Y 35.6638, Z 1.6667, A 0.000, B 0.000, C 0.000 }
gfCNCPoint1[7988] = {X -8.0008, Y 35.6638, Z 11.0000, A 0.000, B 0.000, C 0.000 }
gfCNCPoint1[7989] = {X -7.6965, Y 17.3004, Z 11.0000, A 0.000, B 0.000, C 0.000 }
gfCNCPoint1[7990] = {X -7.6965, Y 17.3004, Z 1.6667, A 0.000, B 0.000, C 0.000 }
gfCNCPoint1[7991] = {X -7.6965, Y 17.3004, Z -1.3333, A 0.000, B 0.000, C 0.000 }
gfCNCPoint1[7992] = {X -4.2198, Y 17.3004, Z -1.3333, A 0.000, B 0.000, C 0.000 }
gfCNCPoint1[7993] = {X -3.6965, Y 13.3348, Z -1.3333, A 0.000, B 0.000, C 0.000 }
gfCNCPoint1[7994] = {X -3.6094, Y 12.8759, Z -1.3333, A 0.000, B 0.000, C 0.000 }
gfCNCPoint1[7995] = {X -3.4715, Y 12.4296, Z -1.3333, A 0.000, B 0.000, C 0.000 }
gfCNCPoint1[7996] = {X -3.0334, Y 11.5714, Z -1.3333, A 0.000, B 0.000, C 0.000 }
gfCNCPoint1[7997] = {X -2.4096, Y 10.8370, Z -1.3333, A 0.000, B 0.000, C 0.000 }
gfCNCPoint1[7998] = {X -1.6337, Y 10.2658, Z -1.3333, A 0.000, B 0.000, C 0.000 }
gfCNCPoint1[7999] = {X -1.0364, Y 9.9251, Z -1.3333, A 0.000, B 0.000, C 0.000 }
gfCNCPoint1[8000] = {X -0.1655, Y 9.5524, Z -1.3333, A 0.000, B 0.000, C 0.000 }
gfCNCPoint1[8001] = {X 0.7672, Y 9.3865, Z -1.3333, A 0.000, B 0.000, C 0.000 }
gfCNCPoint1[8002] = {X 1.7132, Y 9.4358, Z -1.3333, A 0.000, B 0.000, C 0.000 }
gfCNCPoint1[8003] = {X 2.6235, Y 9.6979, Z -1.3333, A 0.000, B 0.000, C 0.000 }
gfCNCPoint1[8004] = {X 3.4270, Y 9.3205, Z -1.3333, A 0.000, B 0.000, C 0.000 }
gfCNCPoint1[8005] = {X 4.2527, Y 8.9949, Z -1.3333, A 0.000, B 0.000, C 0.000 }
gfCNCPoint1[8006] = {X 6.1511, Y 8.3302, Z -1.3333, A 0.000, B 0.000, C 0.000 }
gfCNCPoint1[8007] = {X 8.0998, Y 7.8318, Z -1.3333, A 0.000, B 0.000, C 0.000 }
gfCNCPoint1[8008] = {X 10.0841, Y 7.5033, Z -1.3333, A 0.000, B 0.000, C 0.000 }
gfCNCPoint1[8009] = {X 12.0895, Y 7.3472, Z -1.3333, A 0.000, B 0.000, C 0.000 }
gfCNCPoint1[8010] = {X 14.1008, Y 7.3646, Z -1.3333, A 0.000, B 0.000, C 0.000 }
gfCNCPoint1[8011] = {X 16.1031, Y 7.5554, Z -1.3333, A 0.000, B 0.000, C 0.000 }
gfCNCPoint1[8012] = {X 17.9097, Y 7.8860, Z -1.3333, A 0.000, B 0.000, C 0.000 }
gfCNCPoint1[8013] = {X 19.6711, Y 8.4063, Z -1.3333, A 0.000, B 0.000, C 0.000 }
gfCNCPoint1[8014] = {X 21.3675, Y 9.1103, Z -1.3333, A 0.000, B 0.000, C 0.000 }
gfCNCPoint1[8015] = {X 22.9796, Y 9.9903, Z -1.3333, A 0.000, B 0.000, C 0.000 }
gfCNCPoint1[8016] = {X 24.4894, Y 11.0362, Z -1.3333, A 0.000, B 0.000, C 0.000 }
gfCNCPoint1[8017] = {X 25.5604, Y 11.9735, Z -1.3333, A 0.000, B 0.000, C 0.000 }
gfCNCPoint1[8018] = {X 26.5213, Y 13.0234, Z -1.3333, A 0.000, B 0.000, C 0.000 }
gfCNCPoint1[8019] = {X 27.3603, Y 14.1732, Z -1.3333, A 0.000, B 0.000, C 0.000 }
gfCNCPoint1[8020] = {X 28.0670, Y 15.4087, Z -1.3333, A 0.000, B 0.000, C 0.000 }
gfCNCPoint1[8021] = {X 28.6327, Y 16.7147, Z -1.3333, A 0.000, B 0.000, C 0.000 }
gfCNCPoint1[8022] = {X 29.1015, Y 18.3531, Z -1.3333, A 0.000, B 0.000, C 0.000 }
gfCNCPoint1[8023] = {X 29.3796, Y 20.0345, Z -1.3333, A 0.000, B 0.000, C 0.000 }
gfCNCPoint1[8024] = {X 29.4635, Y 21.7366, Z -1.3333, A 0.000, B 0.000, C 0.000 }
gfCNCPoint1[8025] = {X 29.3521, Y 23.4372, Z -1.3333, A 0.000, B 0.000, C 0.000 }
gfCNCPoint1[8026] = {X 29.0467, Y 25.1138, Z -1.3333, A 0.000, B 0.000, C 0.000 }
gfCNCPoint1[8027] = {X 28.5886, Y 26.5986, Z -1.3333, A 0.000, B 0.000, C 0.000 }
gfCNCPoint1[8028] = {X 27.9349, Y 28.0082, Z -1.3333, A 0.000, B 0.000, C 0.000 }
gfCNCPoint1[8029] = {X 27.0975, Y 29.3172, Z -1.3333, A 0.000, B 0.000, C 0.000 }
gfCNCPoint1[8030] = {X 26.0917, Y 30.5016, Z -1.3333, A 0.000, B 0.000, C 0.000 }
gfCNCPoint1[8031] = {X 24.9358, Y 31.5399, Z -1.3333, A 0.000, B 0.000, C 0.000 }
gfCNCPoint1[8032] = {X 25.1514, Y 31.5958, Z -1.3333, A 0.000, B 0.000, C 0.000 }
gfCNCPoint1[8033] = {X 25.3638, Y 31.6632, Z -1.3333, A 0.000, B 0.000, C 0.000 }
gfCNCPoint1[8034] = {X 26.0973, Y 32.0006, Z -1.3333, A 0.000, B 0.000, C 0.000 }
gfCNCPoint1[8035] = {X 26.7518, Y 32.4733, Z -1.3333, A 0.000, B 0.000, C 0.000 }
gfCNCPoint1[8036] = {X 27.3027, Y 33.0635, Z -1.3333, A 0.000, B 0.000, C 0.000 }
gfCNCPoint1[8037] = {X 27.7292, Y 33.7491, Z -1.3333, A 0.000, B 0.000, C 0.000 }
gfCNCPoint1[8038] = {X 30.7660, Y 40.0227, Z -1.3333, A 0.000, B 0.000, C 0.000 }
gfCNCPoint1[8039] = {X 31.0747, Y 40.8982, Z -1.3333, A 0.000, B 0.000, C 0.000 }
gfCNCPoint1[8040] = {X 31.1815, Y 41.8203, Z -1.3333, A 0.000, B 0.000, C 0.000 }
gfCNCPoint1[8041] = {X 31.0813, Y 42.7431, Z -1.3333, A 0.000, B 0.000, C 0.000 }
gfCNCPoint1[8042] = {X 30.7789, Y 43.6208, Z -1.3333, A 0.000, B 0.000, C 0.000 }
gfCNCPoint1[8043] = {X 30.2893, Y 44.4095, Z -1.3333, A 0.000, B 0.000, C 0.000 }
gfCNCPoint1[8044] = {X 29.6371, Y 45.0700, Z -1.3333, A 0.000, B 0.000, C 0.000 }
gfCNCPoint1[8045] = {X 29.1009, Y 45.5036, Z -1.3333, A 0.000, B 0.000, C 0.000 }
gfCNCPoint1[8046] = {X 28.4097, Y 45.9559, Z -1.3333, A 0.000, B 0.000, C 0.000 }
gfCNCPoint1[8047] = {X 27.6431, Y 46.2633, Z -1.3333, A 0.000, B 0.000, C 0.000 }
gfCNCPoint1[8048] = {X 26.8309, Y 46.4140, Z -1.3333, A 0.000, B 0.000, C 0.000 }
gfCNCPoint1[8049] = {X 26.0050, Y 46.4020, Z -1.3333, A 0.000, B 0.000, C 0.000 }
gfCNCPoint1[8050] = {X 25.1976, Y 46.2278, Z -1.3333, A 0.000, B 0.000, C 0.000 }
gfCNCPoint1[8051] = {X 23.1719, Y 47.2953, Z -1.3333, A 0.000, B 0.000, C 0.000 }
gfCNCPoint1[8052] = {X 21.0665, Y 48.1954, Z -1.3333, A 0.000, B 0.000, C 0.000 }
gfCNCPoint1[8053] = {X 18.8952, Y 48.9223, Z -1.3333, A 0.000, B 0.000, C 0.000 }
gfCNCPoint1[8054] = {X 18.4031, Y 49.0586, Z -1.3333, A 0.000, B 0.000, C 0.000 }
gfCNCPoint1[8055] = {X 16.5527, Y 49.4867, Z -1.3333, A 0.000, B 0.000, C 0.000 }
gfCNCPoint1[8056] = {X 14.6724, Y 49.7543, Z -1.3333, A 0.000, B 0.000, C 0.000 }
gfCNCPoint1[8057] = {X 12.7761, Y 49.8595, Z -1.3333, A 0.000, B 0.000, C 0.000 }
gfCNCPoint1[8058] = {X 10.8777, Y 49.8015, Z -1.3333, A 0.000, B 0.000, C 0.000 }
gfCNCPoint1[8059] = {X 8.9913, Y 49.5808, Z -1.3333, A 0.000, B 0.000, C 0.000 }
gfCNCPoint1[8060] = {X 7.3795, Y 49.2756, Z -1.3333, A 0.000, B 0.000, C 0.000 }
gfCNCPoint1[8061] = {X 5.8046, Y 48.8161, Z -1.3333, A 0.000, B 0.000, C 0.000 }
gfCNCPoint1[8062] = {X 4.2815, Y 48.2068, Z -1.3333, A 0.000, B 0.000, C 0.000 }
gfCNCPoint1[8063] = {X 2.8244, Y 47.4533, Z -1.3333, A 0.000, B 0.000, C 0.000 }
gfCNCPoint1[8064] = {X 1.4467, Y 46.5626, Z -1.3333, A 0.000, B 0.000, C 0.000 }
gfCNCPoint1[8065] = {X 0.1371, Y 45.5096, Z -1.3333, A 0.000, B 0.000, C 0.000 }
gfCNCPoint1[8066] = {X -1.0269, Y 44.2977, Z -1.3333, A 0.000, B 0.000, C 0.000 }
gfCNCPoint1[8067] = {X -2.0263, Y 42.9468, Z -1.3333, A 0.000, B 0.000, C 0.000 }
gfCNCPoint1[8068] = {X -2.8446, Y 41.4791, Z -1.3333, A 0.000, B 0.000, C 0.000 }
gfCNCPoint1[8069] = {X -3.4683, Y 39.9187, Z -1.3333, A 0.000, B 0.000, C 0.000 }
gfCNCPoint1[8070] = {X -3.5884, Y 39.5314, Z -1.3333, A 0.000, B 0.000, C 0.000 }
gfCNCPoint1[8071] = {X -3.6965, Y 39.1406, Z -1.3333, A 0.000, B 0.000, C 0.000 }
gfCNCPoint1[8072] = {X -4.7025, Y 35.2692, Z -1.3333, A 0.000, B 0.000, C 0.000 }
gfCNCPoint1[8073] = {X -8.0047, Y 35.2647, Z -1.3333, A 0.000, B 0.000, C 0.000 }
gfCNCPoint1[8074] = {X -8.0047, Y 35.2647, Z 1.6667, A 0.000, B 0.000, C 0.000 }
gfCNCPoint1[8075] = {X -8.0047, Y 35.2647, Z 11.0000, A 0.000, B 0.000, C 0.000 }
gfCNCPoint1[8076] = {X -7.9984, Y 34.8133, Z 11.0000, A 0.000, B 0.000, C 0.000 }
gfCNCPoint1[8077] = {X -7.9984, Y 34.8133, Z 1.6667, A 0.000, B 0.000, C 0.000 }
gfCNCPoint1[8078] = {X -7.9984, Y 34.8133, Z -1.3333, A 0.000, B 0.000, C 0.000 }
gfCNCPoint1[8079] = {X -4.8614, Y 34.8955, Z -1.3333, A 0.000, B 0.000, C 0.000 }
gfCNCPoint1[8080] = {X -3.6965, Y 31.0689, Z -1.3333, A 0.000, B 0.000, C 0.000 }
gfCNCPoint1[8081] = {X -3.6589, Y 30.9476, Z -1.3333, A 0.000, B 0.000, C 0.000 }
gfCNCPoint1[8082] = {X -3.6203, Y 30.8265, Z -1.3333, A 0.000, B 0.000, C 0.000 }
gfCNCPoint1[8083] = {X -3.2922, Y 29.9174, Z -1.3333, A 0.000, B 0.000, C 0.000 }
gfCNCPoint1[8084] = {X -2.9041, Y 29.0322, Z -1.3333, A 0.000, B 0.000, C 0.000 }
gfCNCPoint1[8085] = {X -2.2642, Y 27.8859, Z -1.3333, A 0.000, B 0.000, C 0.000 }
gfCNCPoint1[8086] = {X -1.4890, Y 26.8265, Z -1.3333, A 0.000, B 0.000, C 0.000 }
gfCNCPoint1[8087] = {X -0.5901, Y 25.8698, Z -1.3333, A 0.000, B 0.000, C 0.000 }
gfCNCPoint1[8088] = {X 0.4190, Y 25.0301, Z -1.3333, A 0.000, B 0.000, C 0.000 }
gfCNCPoint1[8089] = {X 1.5231, Y 24.3200, Z -1.3333, A 0.000, B 0.000, C 0.000 }
gfCNCPoint1[8090] = {X 1.4461, Y 24.2903, Z -1.3333, A 0.000, B 0.000, C 0.000 }
gfCNCPoint1[8091] = {X 1.3697, Y 24.2592, Z -1.3333, A 0.000, B 0.000, C 0.000 }
gfCNCPoint1[8092] = {X 0.6314, Y 23.8616, Z -1.3333, A 0.000, B 0.000, C 0.000 }
gfCNCPoint1[8093] = {X -0.0162, Y 23.3289, Z -1.3333, A 0.000, B 0.000, C 0.000 }
gfCNCPoint1[8094] = {X -0.5487, Y 22.6811, Z -1.3333, A 0.000, B 0.000, C 0.000 }
gfCNCPoint1[8095] = {X -0.9460, Y 21.9427, Z -1.3333, A 0.000, B 0.000, C 0.000 }
gfCNCPoint1[8096] = {X -3.6215, Y 15.3844, Z -1.3333, A 0.000, B 0.000, C 0.000 }
gfCNCPoint1[8097] = {X -3.6604, Y 15.2751, Z -1.3333, A 0.000, B 0.000, C 0.000 }
gfCNCPoint1[8098] = {X -3.6965, Y 15.1648, Z -1.3333, A 0.000, B 0.000, C 0.000 }
gfCNCPoint1[8099] = {X -4.8869, Y 11.3461, Z -1.3333, A 0.000, B 0.000, C 0.000 }
gfCNCPoint1[8100] = {X -7.6965, Y 11.3461, Z -1.3333, A 0.000, B 0.000, C 0.000 }
gfCNCPoint1[8101] = {X -7.6965, Y 11.3461, Z 1.6667, A 0.000, B 0.000, C 0.000 }
gfCNCPoint1[8102] = {X -7.6965, Y 11.3461, Z 11.0000, A 0.000, B 0.000, C 0.000 }
gfCNCPoint1[8103] = {X -8.0043, Y 35.1810, Z 11.0000, A 0.000, B 0.000, C 0.000 }
gfCNCPoint1[8104] = {X -8.0043, Y 35.1810, Z 1.6667, A 0.000, B 0.000, C 0.000 }
gfCNCPoint1[8105] = {X -8.0043, Y 35.1810, Z -1.3333, A 0.000, B 0.000, C 0.000 }
gfCNCPoint1[8106] = {X -4.7892, Y 35.2002, Z -1.3333, A 0.000, B 0.000, C 0.000 }
gfCNCPoint1[8107] = {X -3.6965, Y 31.3523, Z -1.3333, A 0.000, B 0.000, C 0.000 }
gfCNCPoint1[8108] = {X -3.6226, Y 31.1011, Z -1.3333, A 0.000, B 0.000, C 0.000 }
gfCNCPoint1[8109] = {X -3.5442, Y 30.8512, Z -1.3333, A 0.000, B 0.000, C 0.000 }
gfCNCPoint1[8110] = {X -3.2179, Y 29.9471, Z -1.3333, A 0.000, B 0.000, C 0.000 }
gfCNCPoint1[8111] = {X -2.8320, Y 29.0667, Z -1.3333, A 0.000, B 0.000, C 0.000 }
gfCNCPoint1[8112] = {X -2.1775, Y 27.8990, Z -1.3333, A 0.000, B 0.000, C 0.000 }
gfCNCPoint1[8113] = {X -1.3816, Y 26.8227, Z -1.3333, A 0.000, B 0.000, C 0.000 }
gfCNCPoint1[8114] = {X -0.4569, Y 25.8549, Z -1.3333, A 0.000, B 0.000, C 0.000 }
gfCNCPoint1[8115] = {X 0.5821, Y 25.0109, Z -1.3333, A 0.000, B 0.000, C 0.000 }
gfCNCPoint1[8116] = {X 1.7187, Y 24.3039, Z -1.3333, A 0.000, B 0.000, C 0.000 }
gfCNCPoint1[8117] = {X 1.5585, Y 24.2478, Z -1.3333, A 0.000, B 0.000, C 0.000 }
gfCNCPoint1[8118] = {X 1.4006, Y 24.1854, Z -1.3333, A 0.000, B 0.000, C 0.000 }
gfCNCPoint1[8119] = {X 0.6760, Y 23.7952, Z -1.3333, A 0.000, B 0.000, C 0.000 }
gfCNCPoint1[8120] = {X 0.0404, Y 23.2724, Z -1.3333, A 0.000, B 0.000, C 0.000 }
gfCNCPoint1[8121] = {X -0.4822, Y 22.6366, Z -1.3333, A 0.000, B 0.000, C 0.000 }
gfCNCPoint1[8122] = {X -0.8722, Y 21.9118, Z -1.3333, A 0.000, B 0.000, C 0.000 }
gfCNCPoint1[8123] = {X -3.5465, Y 15.3566, Z -1.3333, A 0.000, B 0.000, C 0.000 }
gfCNCPoint1[8124] = {X -3.6290, Y 15.1121, Z -1.3333, A 0.000, B 0.000, C 0.000 }
gfCNCPoint1[8125] = {X -3.6965, Y 14.8631, Z -1.3333, A 0.000, B 0.000, C 0.000 }
gfCNCPoint1[8126] = {X -4.6248, Y 10.9723, Z -1.3333, A 0.000, B 0.000, C 0.000 }
gfCNCPoint1[8127] = {X -7.6965, Y 10.9723, Z -1.3333, A 0.000, B 0.000, C 0.000 }
gfCNCPoint1[8128] = {X -7.6965, Y 10.9723, Z 1.6667, A 0.000, B 0.000, C 0.000 }
gfCNCPoint1[8129] = {X -7.6965, Y 10.9723, Z 11.0000, A 0.000, B 0.000, C 0.000 }
gfCNCPoint1[8130] = {X -8.0024, Y 35.5776, Z 11.0000, A 0.000, B 0.000, C 0.000 }
gfCNCPoint1[8131] = {X -8.0024, Y 35.5776, Z 1.6667, A 0.000, B 0.000, C 0.000 }
gfCNCPoint1[8132] = {X -8.0024, Y 35.5776, Z -1.3333, A 0.000, B 0.000, C 0.000 }
gfCNCPoint1[8133] = {X -4.7106, Y 35.5254, Z -1.3333, A 0.000, B 0.000, C 0.000 }
gfCNCPoint1[8134] = {X -3.6965, Y 31.6561, Z -1.3333, A 0.000, B 0.000, C 0.000 }
gfCNCPoint1[8135] = {X -3.5878, Y 31.2643, Z -1.3333, A 0.000, B 0.000, C 0.000 }
gfCNCPoint1[8136] = {X -3.4681, Y 30.8758, Z -1.3333, A 0.000, B 0.000, C 0.000 }
gfCNCPoint1[8137] = {X -3.1436, Y 29.9767, Z -1.3333, A 0.000, B 0.000, C 0.000 }
gfCNCPoint1[8138] = {X -2.7598, Y 29.1013, Z -1.3333, A 0.000, B 0.000, C 0.000 }
gfCNCPoint1[8139] = {X -2.0891, Y 27.9097, Z -1.3333, A 0.000, B 0.000, C 0.000 }
gfCNCPoint1[8140] = {X -1.2700, Y 26.8149, Z -1.3333, A 0.000, B 0.000, C 0.000 }
gfCNCPoint1[8141] = {X -0.3164, Y 25.8350, Z -1.3333, A 0.000, B 0.000, C 0.000 }
gfCNCPoint1[8142] = {X 0.7559, Y 24.9866, Z -1.3333, A 0.000, B 0.000, C 0.000 }
gfCNCPoint1[8143] = {X 1.9288, Y 24.2838, Z -1.3333, A 0.000, B 0.000, C 0.000 }
gfCNCPoint1[8144] = {X 1.6774, Y 24.2056, Z -1.3333, A 0.000, B 0.000, C 0.000 }
gfCNCPoint1[8145] = {X 1.4316, Y 24.1116, Z -1.3333, A 0.000, B 0.000, C 0.000 }
gfCNCPoint1[8146] = {X 0.7206, Y 23.7288, Z -1.3333, A 0.000, B 0.000, C 0.000 }
gfCNCPoint1[8147] = {X 0.0970, Y 23.2158, Z -1.3333, A 0.000, B 0.000, C 0.000 }
gfCNCPoint1[8148] = {X -0.4158, Y 22.5920, Z -1.3333, A 0.000, B 0.000, C 0.000 }
gfCNCPoint1[8149] = {X -0.7984, Y 21.8809, Z -1.3333, A 0.000, B 0.000, C 0.000 }
gfCNCPoint1[8150] = {X -3.4715, Y 15.3287, Z -1.3333, A 0.000, B 0.000, C 0.000 }
gfCNCPoint1[8151] = {X -3.6094, Y 14.8824, Z -1.3333, A 0.000, B 0.000, C 0.000 }
gfCNCPoint1[8152] = {X -3.6965, Y 14.4234, Z -1.3333, A 0.000, B 0.000, C 0.000 }
gfCNCPoint1[8153] = {X -4.2198, Y 10.4578, Z -1.3333, A 0.000, B 0.000, C 0.000 }
gfCNCPoint1[8154] = {X -7.6965, Y 10.4578, Z -1.3333, A 0.000, B 0.000, C 0.000 }
gfCNCPoint1[8155] = {X -7.6965, Y 10.4578, Z 1.6667, A 0.000, B 0.000, C 0.000 }
gfCNCPoint1[8156] = {X -7.6965, Y 10.4578, Z 11.0000, A 0.000, B 0.000, C 0.000 }
gfCNCPoint1[8157] = {X -7.9904, Y 36.0104, Z 11.0000, A 0.000, B 0.000, C 0.000 }
gfCNCPoint1[8158] = {X -7.9904, Y 36.0104, Z 1.6667, A 0.000, B 0.000, C 0.000 }
gfCNCPoint1[8159] = {X -7.9904, Y 36.0104, Z -1.3333, A 0.000, B 0.000, C 0.000 }
gfCNCPoint1[8160] = {X -4.6237, Y 35.8767, Z -1.3333, A 0.000, B 0.000, C 0.000 }
gfCNCPoint1[8161] = {X -3.6965, Y 31.9857, Z -1.3333, A 0.000, B 0.000, C 0.000 }
gfCNCPoint1[8162] = {X -3.5550, Y 31.4401, Z -1.3333, A 0.000, B 0.000, C 0.000 }
gfCNCPoint1[8163] = {X -3.3920, Y 30.9005, Z -1.3333, A 0.000, B 0.000, C 0.000 }
gfCNCPoint1[8164] = {X -3.0693, Y 30.0064, Z -1.3333, A 0.000, B 0.000, C 0.000 }
gfCNCPoint1[8165] = {X -2.6877, Y 29.1358, Z -1.3333, A 0.000, B 0.000, C 0.000 }
gfCNCPoint1[8166] = {X -1.9984, Y 27.9173, Z -1.3333, A 0.000, B 0.000, C 0.000 }
gfCNCPoint1[8167] = {X -1.1529, Y 26.8015, Z -1.3333, A 0.000, B 0.000, C 0.000 }
gfCNCPoint1[8168] = {X -0.1663, Y 25.8084, Z -1.3333, A 0.000, B 0.000, C 0.000 }
gfCNCPoint1[8169] = {X 0.9439, Y 24.9556, Z -1.3333, A 0.000, B 0.000, C 0.000 }
gfCNCPoint1[8170] = {X 2.1579, Y 24.2584, Z -1.3333, A 0.000, B 0.000, C 0.000 }
gfCNCPoint1[8171] = {X 1.8053, Y 24.1637, Z -1.3333, A 0.000, B 0.000, C 0.000 }
gfCNCPoint1[8172] = {X 1.4625, Y 24.0378, Z -1.3333, A 0.000, B 0.000, C 0.000 }
gfCNCPoint1[8173] = {X 0.7652, Y 23.6623, Z -1.3333, A 0.000, B 0.000, C 0.000 }
gfCNCPoint1[8174] = {X 0.1536, Y 23.1592, Z -1.3333, A 0.000, B 0.000, C 0.000 }
gfCNCPoint1[8175] = {X -0.3493, Y 22.5474, Z -1.3333, A 0.000, B 0.000, C 0.000 }
gfCNCPoint1[8176] = {X -0.7246, Y 21.8500, Z -1.3333, A 0.000, B 0.000, C 0.000 }
gfCNCPoint1[8177] = {X -3.3965, Y 15.3008, Z -1.3333, A 0.000, B 0.000, C 0.000 }
gfCNCPoint1[8178] = {X -3.6235, Y 14.3620, Z -1.3333, A 0.000, B 0.000, C 0.000 }
gfCNCPoint1[8179] = {X -3.6235, Y 13.3962, Z -1.3333, A 0.000, B 0.000, C 0.000 }
gfCNCPoint1[8180] = {X -3.3965, Y 12.4574, Z -1.3333, A 0.000, B 0.000, C 0.000 }
gfCNCPoint1[8181] = {X -2.9669, Y 11.6157, Z -1.3333, A 0.000, B 0.000, C 0.000 }
gfCNCPoint1[8182] = {X -2.3551, Y 10.8955, Z -1.3333, A 0.000, B 0.000, C 0.000 }
gfCNCPoint1[8183] = {X -1.5940, Y 10.3353, Z -1.3333, A 0.000, B 0.000, C 0.000 }
gfCNCPoint1[8184] = {X -0.9968, Y 9.9946, Z -1.3333, A 0.000, B 0.000, C 0.000 }
gfCNCPoint1[8185] = {X -0.1338, Y 9.6264, Z -1.3333, A 0.000, B 0.000, C 0.000 }
gfCNCPoint1[8186] = {X 0.7905, Y 9.4652, Z -1.3333, A 0.000, B 0.000, C 0.000 }
gfCNCPoint1[8187] = {X 1.7272, Y 9.5194, Z -1.3333, A 0.000, B 0.000, C 0.000 }
gfCNCPoint1[8188] = {X 2.6267, Y 9.7861, Z -1.3333, A 0.000, B 0.000, C 0.000 }
gfCNCPoint1[8189] = {X 3.4423, Y 9.4011, Z -1.3333, A 0.000, B 0.000, C 0.000 }
gfCNCPoint1[8190] = {X 4.2810, Y 9.0697, Z -1.3333, A 0.000, B 0.000, C 0.000 }
gfCNCPoint1[8191] = {X 6.1732, Y 8.4071, Z -1.3333, A 0.000, B 0.000, C 0.000 }
gfCNCPoint1[8192] = {X 8.1154, Y 7.9103, Z -1.3333, A 0.000, B 0.000, C 0.000 }
gfCNCPoint1[8193] = {X 10.0933, Y 7.5828, Z -1.3333, A 0.000, B 0.000, C 0.000 }
gfCNCPoint1[8194] = {X 12.0920, Y 7.4271, Z -1.3333, A 0.000, B 0.000, C 0.000 }
gfCNCPoint1[8195] = {X 14.0967, Y 7.4445, Z -1.3333, A 0.000, B 0.000, C 0.000 }
gfCNCPoint1[8196] = {X 16.0925, Y 7.6347, Z -1.3333, A 0.000, B 0.000, C 0.000 }
gfCNCPoint1[8197] = {X 17.8908, Y 7.9637, Z -1.3333, A 0.000, B 0.000, C 0.000 }
gfCNCPoint1[8198] = {X 19.6442, Y 8.4816, Z -1.3333, A 0.000, B 0.000, C 0.000 }
gfCNCPoint1[8199] = {X 21.3328, Y 9.1824, Z -1.3333, A 0.000, B 0.000, C 0.000 }
gfCNCPoint1[8200] = {X 22.9375, Y 10.0583, Z -1.3333, A 0.000, B 0.000, C 0.000 }
gfCNCPoint1[8201] = {X 24.4404, Y 11.0994, Z -1.3333, A 0.000, B 0.000, C 0.000 }
gfCNCPoint1[8202] = {X 25.5046, Y 12.0308, Z -1.3333, A 0.000, B 0.000, C 0.000 }
gfCNCPoint1[8203] = {X 26.4594, Y 13.0740, Z -1.3333, A 0.000, B 0.000, C 0.000 }
gfCNCPoint1[8204] = {X 27.2930, Y 14.2165, Z -1.3333, A 0.000, B 0.000, C 0.000 }
gfCNCPoint1[8205] = {X 27.9952, Y 15.4440, Z -1.3333, A 0.000, B 0.000, C 0.000 }
gfCNCPoint1[8206] = {X 28.5574, Y 16.7417, Z -1.3333, A 0.000, B 0.000, C 0.000 }
gfCNCPoint1[8207] = {X 29.0236, Y 18.3713, Z -1.3333, A 0.000, B 0.000, C 0.000 }
gfCNCPoint1[8208] = {X 29.3001, Y 20.0435, Z -1.3333, A 0.000, B 0.000, C 0.000 }
gfCNCPoint1[8209] = {X 29.3835, Y 21.7364, Z -1.3333, A 0.000, B 0.000, C 0.000 }
gfCNCPoint1[8210] = {X 29.2726, Y 23.4277, Z -1.3333, A 0.000, B 0.000, C 0.000 }
gfCNCPoint1[8211] = {X 28.9689, Y 25.0951, Z -1.3333, A 0.000, B 0.000, C 0.000 }
gfCNCPoint1[8212] = {X 28.5015, Y 26.6020, Z -1.3333, A 0.000, B 0.000, C 0.000 }
gfCNCPoint1[8213] = {X 27.8313, Y 28.0303, Z -1.3333, A 0.000, B 0.000, C 0.000 }
gfCNCPoint1[8214] = {X 26.9711, Y 29.3528, Z -1.3333, A 0.000, B 0.000, C 0.000 }
gfCNCPoint1[8215] = {X 25.9372, Y 30.5445, Z -1.3333, A 0.000, B 0.000, C 0.000 }
gfCNCPoint1[8216] = {X 24.7493, Y 31.5827, Z -1.3333, A 0.000, B 0.000, C 0.000 }
gfCNCPoint1[8217] = {X 25.0463, Y 31.6498, Z -1.3333, A 0.000, B 0.000, C 0.000 }
gfCNCPoint1[8218] = {X 25.3375, Y 31.7388, Z -1.3333, A 0.000, B 0.000, C 0.000 }
gfCNCPoint1[8219] = {X 26.0569, Y 32.0696, Z -1.3333, A 0.000, B 0.000, C 0.000 }
gfCNCPoint1[8220] = {X 26.6989, Y 32.5333, Z -1.3333, A 0.000, B 0.000, C 0.000 }
gfCNCPoint1[8221] = {X 27.2392, Y 33.1122, Z -1.3333, A 0.000, B 0.000, C 0.000 }
gfCNCPoint1[8222] = {X 27.6575, Y 33.7845, Z -1.3333, A 0.000, B 0.000, C 0.000 }
gfCNCPoint1[8223] = {X 30.6940, Y 40.0576, Z -1.3333, A 0.000, B 0.000, C 0.000 }
gfCNCPoint1[8224] = {X 30.9967, Y 40.9162, Z -1.3333, A 0.000, B 0.000, C 0.000 }
gfCNCPoint1[8225] = {X 31.1015, Y 41.8206, Z -1.3333, A 0.000, B 0.000, C 0.000 }
gfCNCPoint1[8226] = {X 31.0032, Y 42.7257, Z -1.3333, A 0.000, B 0.000, C 0.000 }
gfCNCPoint1[8227] = {X 30.7066, Y 43.5864, Z -1.3333, A 0.000, B 0.000, C 0.000 }
gfCNCPoint1[8228] = {X 30.2265, Y 44.3600, Z -1.3333, A 0.000, B 0.000, C 0.000 }
gfCNCPoint1[8229] = {X 29.5868, Y 45.0078, Z -1.3333, A 0.000, B 0.000, C 0.000 }
gfCNCPoint1[8230] = {X 29.0507, Y 45.4413, Z -1.3333, A 0.000, B 0.000, C 0.000 }
gfCNCPoint1[8231] = {X 28.3664, Y 45.8882, Z -1.3333, A 0.000, B 0.000, C 0.000 }
gfCNCPoint1[8232] = {X 27.6071, Y 46.1904, Z -1.3333, A 0.000, B 0.000, C 0.000 }
gfCNCPoint1[8233] = {X 26.8030, Y 46.3360, Z -1.3333, A 0.000, B 0.000, C 0.000 }
gfCNCPoint1[8234] = {X 25.9859, Y 46.3192, Z -1.3333, A 0.000, B 0.000, C 0.000 }
gfCNCPoint1[8235] = {X 25.1884, Y 46.1406, Z -1.3333, A 0.000, B 0.000, C 0.000 }
gfCNCPoint1[8236] = {X 23.1592, Y 47.2127, Z -1.3333, A 0.000, B 0.000, C 0.000 }
gfCNCPoint1[8237] = {X 21.0495, Y 48.1163, Z -1.3333, A 0.000, B 0.000, C 0.000 }
gfCNCPoint1[8238] = {X 18.8733, Y 48.8453, Z -1.3333, A 0.000, B 0.000, C 0.000 }
gfCNCPoint1[8239] = {X 18.3818, Y 48.9815, Z -1.3333, A 0.000, B 0.000, C 0.000 }
gfCNCPoint1[8240] = {X 16.5381, Y 49.4080, Z -1.3333, A 0.000, B 0.000, C 0.000 }
gfCNCPoint1[8241] = {X 14.6646, Y 49.6747, Z -1.3333, A 0.000, B 0.000, C 0.000 }
gfCNCPoint1[8242] = {X 12.7751, Y 49.7795, Z -1.3333, A 0.000, B 0.000, C 0.000 }
gfCNCPoint1[8243] = {X 10.8836, Y 49.7217, Z -1.3333, A 0.000, B 0.000, C 0.000 }
gfCNCPoint1[8244] = {X 9.0040, Y 49.5018, Z -1.3333, A 0.000, B 0.000, C 0.000 }
gfCNCPoint1[8245] = {X 8.2871, Y 49.3865, Z -1.3333, A 0.000, B 0.000, C 0.000 }
gfCNCPoint1[8246] = {X 6.4792, Y 48.9501, Z -1.3333, A 0.000, B 0.000, C 0.000 }
gfCNCPoint1[8247] = {X 4.7303, Y 48.3177, Z -1.3333, A 0.000, B 0.000, C 0.000 }
gfCNCPoint1[8248] = {X 3.0615, Y 47.4968, Z -1.3333, A 0.000, B 0.000, C 0.000 }
gfCNCPoint1[8249] = {X 1.4931, Y 46.4974, Z -1.3333, A 0.000, B 0.000, C 0.000 }
gfCNCPoint1[8250] = {X 0.1914, Y 45.4508, Z -1.3333, A 0.000, B 0.000, C 0.000 }
gfCNCPoint1[8251] = {X -0.9656, Y 44.2463, Z -1.3333, A 0.000, B 0.000, C 0.000 }
gfCNCPoint1[8252] = {X -1.9590, Y 42.9035, Z -1.3333, A 0.000, B 0.000, C 0.000 }
gfCNCPoint1[8253] = {X -2.7723, Y 41.4447, Z -1.3333, A 0.000, B 0.000, C 0.000 }
gfCNCPoint1[8254] = {X -3.3923, Y 39.8938, Z -1.3333, A 0.000, B 0.000, C 0.000 }
gfCNCPoint1[8255] = {X -3.5562, Y 39.3535, Z -1.3333, A 0.000, B 0.000, C 0.000 }
gfCNCPoint1[8256] = {X -3.6965, Y 38.8066, Z -1.3333, A 0.000, B 0.000, C 0.000 }
gfCNCPoint1[8257] = {X -4.6061, Y 34.9114, Z -1.3333, A 0.000, B 0.000, C 0.000 }
gfCNCPoint1[8258] = {X -7.9987, Y 34.8246, Z -1.3333, A 0.000, B 0.000, C 0.000 }
gfCNCPoint1[8259] = {X -7.9987, Y 34.8246, Z 1.6667, A 0.000, B 0.000, C 0.000 }
gfCNCPoint1[8260] = {X -7.9987, Y 34.8246, Z 11.0000, A 0.000, B 0.000, C 0.000 }
gfCNCPoint1[8261] = {X -7.9649, Y 36.4908, Z 11.0000, A 0.000, B 0.000, C 0.000 }
gfCNCPoint1[8262] = {X -7.9649, Y 36.4908, Z 1.6667, A 0.000, B 0.000, C 0.000 }
gfCNCPoint1[8263] = {X -7.9649, Y 36.4908, Z -1.3333, A 0.000, B 0.000, C 0.000 }
gfCNCPoint1[8264] = {X -4.5262, Y 36.2629, Z -1.3333, A 0.000, B 0.000, C 0.000 }
gfCNCPoint1[8265] = {X -3.6965, Y 32.3499, Z -1.3333, A 0.000, B 0.000, C 0.000 }
gfCNCPoint1[8266] = {X -3.5247, Y 31.6325, Z -1.3333, A 0.000, B 0.000, C 0.000 }
gfCNCPoint1[8267] = {X -3.3159, Y 30.9251, Z -1.3333, A 0.000, B 0.000, C 0.000 }
gfCNCPoint1[8268] = {X -2.9950, Y 30.0360, Z -1.3333, A 0.000, B 0.000, C 0.000 }
gfCNCPoint1[8269] = {X -2.6155, Y 29.1703, Z -1.3333, A 0.000, B 0.000, C 0.000 }
gfCNCPoint1[8270] = {X -1.9046, Y 27.9204, Z -1.3333, A 0.000, B 0.000, C 0.000 }
gfCNCPoint1[8271] = {X -1.0280, Y 26.7804, Z -1.3333, A 0.000, B 0.000, C 0.000 }
gfCNCPoint1[8272] = {X -0.0026, Y 25.7722, Z -1.3333, A 0.000, B 0.000, C 0.000 }
gfCNCPoint1[8273] = {X 1.1521, Y 24.9152, Z -1.3333, A 0.000, B 0.000, C 0.000 }
gfCNCPoint1[8274] = {X 2.4140, Y 24.2256, Z -1.3333, A 0.000, B 0.000, C 0.000 }
gfCNCPoint1[8275] = {X 1.9458, Y 24.1224, Z -1.3333, A 0.000, B 0.000, C 0.000 }
gfCNCPoint1[8276] = {X 1.4934, Y 23.9640, Z -1.3333, A 0.000, B 0.000, C 0.000 }
gfCNCPoint1[8277] = {X 0.8025, Y 23.5910, Z -1.3333, A 0.000, B 0.000, C 0.000 }
gfCNCPoint1[8278] = {X 0.1977, Y 23.0902, Z -1.3333, A 0.000, B 0.000, C 0.000 }
gfCNCPoint1[8279] = {X -0.2975, Y 22.4809, Z -1.3333, A 0.000, B 0.000, C 0.000 }
gfCNCPoint1[8280] = {X -0.6642, Y 21.7866, Z -1.3333, A 0.000, B 0.000, C 0.000 }
gfCNCPoint1[8281] = {X -3.2754, Y 15.3911, Z -1.3333, A 0.000, B 0.000, C 0.000 }
gfCNCPoint1[8282] = {X -3.2990, Y 15.3322, Z -1.3333, A 0.000, B 0.000, C 0.000 }
gfCNCPoint1[8283] = {X -3.3215, Y 15.2729, Z -1.3333, A 0.000, B 0.000, C 0.000 }
gfCNCPoint1[8284] = {X -3.5441, Y 14.3526, Z -1.3333, A 0.000, B 0.000, C 0.000 }
gfCNCPoint1[8285] = {X -3.5441, Y 13.4057, Z -1.3333, A 0.000, B 0.000, C 0.000 }
gfCNCPoint1[8286] = {X -3.3215, Y 12.4853, Z -1.3333, A 0.000, B 0.000, C 0.000 }
gfCNCPoint1[8287] = {X -2.9003, Y 11.6601, Z -1.3333, A 0.000, B 0.000, C 0.000 }
gfCNCPoint1[8288] = {X -2.3005, Y 10.9540, Z -1.3333, A 0.000, B 0.000, C 0.000 }
gfCNCPoint1[8289] = {X -1.5544, Y 10.4048, Z -1.3333, A 0.000, B 0.000, C 0.000 }
gfCNCPoint1[8290] = {X -0.9063, Y 10.0355, Z -1.3333, A 0.000, B 0.000, C 0.000 }
gfCNCPoint1[8291] = {X -0.0600, Y 9.6884, Z -1.3333, A 0.000, B 0.000, C 0.000 }
gfCNCPoint1[8292] = {X 0.8429, Y 9.5426, Z -1.3333, A 0.000, B 0.000, C 0.000 }
gfCNCPoint1[8293] = {X 1.7554, Y 9.6057, Z -1.3333, A 0.000, B 0.000, C 0.000 }
gfCNCPoint1[8294] = {X 2.6297, Y 9.8745, Z -1.3333, A 0.000, B 0.000, C 0.000 }
gfCNCPoint1[8295] = {X 2.7102, Y 9.8333, Z -1.3333, A 0.000, B 0.000, C 0.000 }
gfCNCPoint1[8296] = {X 2.7910, Y 9.7926, Z -1.3333, A 0.000, B 0.000, C 0.000 }
gfCNCPoint1[8297] = {X 3.5437, Y 9.4444, Z -1.3333, A 0.000, B 0.000, C 0.000 }
gfCNCPoint1[8298] = {X 4.3160, Y 9.1419, Z -1.3333, A 0.000, B 0.000, C 0.000 }
gfCNCPoint1[8299] = {X 6.2009, Y 8.4823, Z -1.3333, A 0.000, B 0.000, C 0.000 }
gfCNCPoint1[8300] = {X 8.1357, Y 7.9877, Z -1.3333, A 0.000, B 0.000, C 0.000 }
gfCNCPoint1[8301] = {X 10.1060, Y 7.6618, Z -1.3333, A 0.000, B 0.000, C 0.000 }
gfCNCPoint1[8302] = {X 12.0970, Y 7.5070, Z -1.3333, A 0.000, B 0.000, C 0.000 }
gfCNCPoint1[8303] = {X 14.0940, Y 7.5244, Z -1.3333, A 0.000, B 0.000, C 0.000 }
gfCNCPoint1[8304] = {X 16.0820, Y 7.7140, Z -1.3333, A 0.000, B 0.000, C 0.000 }
gfCNCPoint1[8305] = {X 16.4805, Y 7.7686, Z -1.3333, A 0.000, B 0.000, C 0.000 }
gfCNCPoint1[8306] = {X 18.1846, Y 8.1180, Z -1.3333, A 0.000, B 0.000, C 0.000 }
gfCNCPoint1[8307] = {X 19.8445, Y 8.6383, Z -1.3333, A 0.000, B 0.000, C 0.000 }
gfCNCPoint1[8308] = {X 21.4431, Y 9.3242, Z -1.3333, A 0.000, B 0.000, C 0.000 }
gfCNCPoint1[8309] = {X 22.9639, Y 10.1685, Z -1.3333, A 0.000, B 0.000, C 0.000 }
gfCNCPoint1[8310] = {X 24.3914, Y 11.1626, Z -1.3333, A 0.000, B 0.000, C 0.000 }
gfCNCPoint1[8311] = {X 25.4488, Y 12.0881, Z -1.3333, A 0.000, B 0.000, C 0.000 }
gfCNCPoint1[8312] = {X 26.3974, Y 13.1246, Z -1.3333, A 0.000, B 0.000, C 0.000 }
gfCNCPoint1[8313] = {X 27.2257, Y 14.2597, Z -1.3333, A 0.000, B 0.000, C 0.000 }
gfCNCPoint1[8314] = {X 27.9235, Y 15.4794, Z -1.3333, A 0.000, B 0.000, C 0.000 }
gfCNCPoint1[8315] = {X 28.4821, Y 16.7687, Z -1.3333, A 0.000, B 0.000, C 0.000 }
gfCNCPoint1[8316] = {X 28.9457, Y 18.3896, Z -1.3333, A 0.000, B 0.000, C 0.000 }
gfCNCPoint1[8317] = {X 29.2207, Y 20.0530, Z -1.3333, A 0.000, B 0.000, C 0.000 }
gfCNCPoint1[8318] = {X 29.3035, Y 21.7368, Z -1.3333, A 0.000, B 0.000, C 0.000 }
gfCNCPoint1[8319] = {X 29.1931, Y 23.4191, Z -1.3333, A 0.000, B 0.000, C 0.000 }
gfCNCPoint1[8320] = {X 28.8909, Y 25.0776, Z -1.3333, A 0.000, B 0.000, C 0.000 }
gfCNCPoint1[8321] = {X 28.4130, Y 26.6088, Z -1.3333, A 0.000, B 0.000, C 0.000 }
gfCNCPoint1[8322] = {X 27.7244, Y 28.0574, Z -1.3333, A 0.000, B 0.000, C 0.000 }
gfCNCPoint1[8323] = {X 26.8387, Y 29.3947, Z -1.3333, A 0.000, B 0.000, C 0.000 }
gfCNCPoint1[8324] = {X 25.7736, Y 30.5940, Z -1.3333, A 0.000, B 0.000, C 0.000 }
gfCNCPoint1[8325] = {X 24.5503, Y 31.6314, Z -1.3333, A 0.000, B 0.000, C 0.000 }
gfCNCPoint1[8326] = {X 24.9353, Y 31.7042, Z -1.3333, A 0.000, B 0.000, C 0.000 }
gfCNCPoint1[8327] = {X 25.3113, Y 31.8143, Z -1.3333, A 0.000, B 0.000, C 0.000 }
gfCNCPoint1[8328] = {X 26.0240, Y 32.1431, Z -1.3333, A 0.000, B 0.000, C 0.000 }
gfCNCPoint1[8329] = {X 26.6588, Y 32.6047, Z -1.3333, A 0.000, B 0.000, C 0.000 }
gfCNCPoint1[8330] = {X 27.1913, Y 33.1813, Z -1.3333, A 0.000, B 0.000, C 0.000 }
gfCNCPoint1[8331] = {X 27.6008, Y 33.8508, Z -1.3333, A 0.000, B 0.000, C 0.000 }
gfCNCPoint1[8332] = {X 30.6220, Y 40.0925, Z -1.3333, A 0.000, B 0.000, C 0.000 }
gfCNCPoint1[8333] = {X 30.9188, Y 40.9342, Z -1.3333, A 0.000, B 0.000, C 0.000 }
gfCNCPoint1[8334] = {X 31.0215, Y 41.8209, Z -1.3333, A 0.000, B 0.000, C 0.000 }
gfCNCPoint1[8335] = {X 30.9251, Y 42.7082, Z -1.3333, A 0.000, B 0.000, C 0.000 }
gfCNCPoint1[8336] = {X 30.6343, Y 43.5521, Z -1.3333, A 0.000, B 0.000, C 0.000 }
gfCNCPoint1[8337] = {X 30.1637, Y 44.3105, Z -1.3333, A 0.000, B 0.000, C 0.000 }
gfCNCPoint1[8338] = {X 29.5365, Y 44.9456, Z -1.3333, A 0.000, B 0.000, C 0.000 }
gfCNCPoint1[8339] = {X 29.0005, Y 45.3790, Z -1.3333, A 0.000, B 0.000, C 0.000 }
gfCNCPoint1[8340] = {X 28.3232, Y 45.8205, Z -1.3333, A 0.000, B 0.000, C 0.000 }
gfCNCPoint1[8341] = {X 27.5713, Y 46.1174, Z -1.3333, A 0.000, B 0.000, C 0.000 }
gfCNCPoint1[8342] = {X 26.7751, Y 46.2579, Z -1.3333, A 0.000, B 0.000, C 0.000 }
gfCNCPoint1[8343] = {X 25.9670, Y 46.2362, Z -1.3333, A 0.000, B 0.000, C 0.000 }
gfCNCPoint1[8344] = {X 25.1795, Y 46.0532, Z -1.3333, A 0.000, B 0.000, C 0.000 }
gfCNCPoint1[8345] = {X 25.1036, Y 46.0973, Z -1.3333, A 0.000, B 0.000, C 0.000 }
gfCNCPoint1[8346] = {X 25.0276, Y 46.1412, Z -1.3333, A 0.000, B 0.000, C 0.000 }
gfCNCPoint1[8347] = {X 23.0410, Y 47.1803, Z -1.3333, A 0.000, B 0.000, C 0.000 }
gfCNCPoint1[8348] = {X 20.9779, Y 48.0579, Z -1.3333, A 0.000, B 0.000, C 0.000 }
gfCNCPoint1[8349] = {X 18.8515, Y 48.7683, Z -1.3333, A 0.000, B 0.000, C 0.000 }
gfCNCPoint1[8350] = {X 18.3604, Y 48.9044, Z -1.3333, A 0.000, B 0.000, C 0.000 }
gfCNCPoint1[8351] = {X 16.5234, Y 49.3294, Z -1.3333, A 0.000, B 0.000, C 0.000 }
gfCNCPoint1[8352] = {X 14.6567, Y 49.5951, Z -1.3333, A 0.000, B 0.000, C 0.000 }
gfCNCPoint1[8353] = {X 12.7741, Y 49.6995, Z -1.3333, A 0.000, B 0.000, C 0.000 }
gfCNCPoint1[8354] = {X 10.8894, Y 49.6420, Z -1.3333, A 0.000, B 0.000, C 0.000 }
gfCNCPoint1[8355] = {X 9.0167, Y 49.4228, Z -1.3333, A 0.000, B 0.000, C 0.000 }
gfCNCPoint1[8356] = {X 8.3007, Y 49.3077, Z -1.3333, A 0.000, B 0.000, C 0.000 }
gfCNCPoint1[8357] = {X 6.5011, Y 48.8732, Z -1.3333, A 0.000, B 0.000, C 0.000 }
gfCNCPoint1[8358] = {X 4.7602, Y 48.2434, Z -1.3333, A 0.000, B 0.000, C 0.000 }
gfCNCPoint1[8359] = {X 3.0991, Y 47.4261, Z -1.3333, A 0.000, B 0.000, C 0.000 }
gfCNCPoint1[8360] = {X 1.5379, Y 46.4312, Z -1.3333, A 0.000, B 0.000, C 0.000 }
gfCNCPoint1[8361] = {X 0.2446, Y 45.3911, Z -1.3333, A 0.000, B 0.000, C 0.000 }
gfCNCPoint1[8362] = {X -0.9051, Y 44.1940, Z -1.3333, A 0.000, B 0.000, C 0.000 }
gfCNCPoint1[8363] = {X -1.8921, Y 42.8597, Z -1.3333, A 0.000, B 0.000, C 0.000 }
gfCNCPoint1[8364] = {X -2.7002, Y 41.4101, Z -1.3333, A 0.000, B 0.000, C 0.000 }
gfCNCPoint1[8365] = {X -3.3163, Y 39.8689, Z -1.3333, A 0.000, B 0.000, C 0.000 }
gfCNCPoint1[8366] = {X -3.5270, Y 39.1560, Z -1.3333, A 0.000, B 0.000, C 0.000 }
gfCNCPoint1[8367] = {X -3.6965, Y 38.4322, Z -1.3333, A 0.000, B 0.000, C 0.000 }
gfCNCPoint1[8368] = {X -4.4960, Y 34.5129, Z -1.3333, A 0.000, B 0.000, C 0.000 }
gfCNCPoint1[8369] = {X -7.9792, Y 34.3285, Z -1.3333, A 0.000, B 0.000, C 0.000 }
gfCNCPoint1[8370] = {X -7.9792, Y 34.3285, Z 1.6667, A 0.000, B 0.000, C 0.000 }
gfCNCPoint1[8371] = {X -7.9792, Y 34.3285, Z 11.0000, A 0.000, B 0.000, C 0.000 }
gfCNCPoint1[8372] = {X 39.8256, Y 26.3831, Z 11.0000, A 0.000, B 0.000, C 0.000 }
gfCNCPoint1[8373] = {X 39.8256, Y 26.3831, Z 1.6667, A 0.000, B 0.000, C 0.000 }
gfCNCPoint1[8374] = {X 39.8256, Y 26.3831, Z -1.3333, A 0.000, B 0.000, C 0.000 }
gfCNCPoint1[8375] = {X 43.6491, Y 27.8070, Z -1.3333, A 0.000, B 0.000, C 0.000 }
gfCNCPoint1[8376] = {X 48.2902, Y 15.3446, Z -1.3333, A 0.000, B 0.000, C 0.000 }
gfCNCPoint1[8377] = {X 47.9078, Y 14.6186, Z -1.3333, A 0.000, B 0.000, C 0.000 }
gfCNCPoint1[8378] = {X 47.6697, Y 13.8333, Z -1.3333, A 0.000, B 0.000, C 0.000 }
gfCNCPoint1[8379] = {X 47.5844, Y 13.0172, Z -1.3333, A 0.000, B 0.000, C 0.000 }
gfCNCPoint1[8380] = {X 47.5842, Y 12.1868, Z -1.3333, A 0.000, B 0.000, C 0.000 }
gfCNCPoint1[8381] = {X 47.6925, Y 11.2255, Z -1.3333, A 0.000, B 0.000, C 0.000 }
gfCNCPoint1[8382] = {X 48.0120, Y 10.3125, Z -1.3333, A 0.000, B 0.000, C 0.000 }
gfCNCPoint1[8383] = {X 48.5267, Y 9.4933, Z -1.3333, A 0.000, B 0.000, C 0.000 }
gfCNCPoint1[8384] = {X 49.2107, Y 8.8093, Z -1.3333, A 0.000, B 0.000, C 0.000 }
gfCNCPoint1[8385] = {X 50.0298, Y 8.2946, Z -1.3333, A 0.000, B 0.000, C 0.000 }
gfCNCPoint1[8386] = {X 50.9429, Y 7.9751, Z -1.3333, A 0.000, B 0.000, C 0.000 }
gfCNCPoint1[8387] = {X 51.9042, Y 7.8668, Z -1.3333, A 0.000, B 0.000, C 0.000 }
gfCNCPoint1[8388] = {X 59.6221, Y 7.8668, Z -1.3333, A 0.000, B 0.000, C 0.000 }
gfCNCPoint1[8389] = {X 60.5834, Y 7.9751, Z -1.3333, A 0.000, B 0.000, C 0.000 }
gfCNCPoint1[8390] = {X 61.4965, Y 8.2946, Z -1.3333, A 0.000, B 0.000, C 0.000 }
gfCNCPoint1[8391] = {X 62.3156, Y 8.8093, Z -1.3333, A 0.000, B 0.000, C 0.000 }
gfCNCPoint1[8392] = {X 62.9996, Y 9.4933, Z -1.3333, A 0.000, B 0.000, C 0.000 }
gfCNCPoint1[8393] = {X 63.5143, Y 10.3124, Z -1.3333, A 0.000, B 0.000, C 0.000 }
gfCNCPoint1[8394] = {X 63.8338, Y 11.2255, Z -1.3333, A 0.000, B 0.000, C 0.000 }
gfCNCPoint1[8395] = {X 63.9421, Y 12.1868, Z -1.3333, A 0.000, B 0.000, C 0.000 }
gfCNCPoint1[8396] = {X 63.9421, Y 12.9781, Z -1.3333, A 0.000, B 0.000, C 0.000 }
gfCNCPoint1[8397] = {X 63.8583, Y 13.8249, Z -1.3333, A 0.000, B 0.000, C 0.000 }
gfCNCPoint1[8398] = {X 63.6101, Y 14.6388, Z -1.3333, A 0.000, B 0.000, C 0.000 }
gfCNCPoint1[8399] = {X 63.2072, Y 15.3883, Z -1.3333, A 0.000, B 0.000, C 0.000 }
gfCNCPoint1[8400] = {X 63.4697, Y 16.0738, Z -1.3333, A 0.000, B 0.000, C 0.000 }
gfCNCPoint1[8401] = {X 66.0338, Y 22.8875, Z -1.3333, A 0.000, B 0.000, C 0.000 }
gfCNCPoint1[8402] = {X 72.2084, Y 39.5004, Z -1.3333, A 0.000, B 0.000, C 0.000 }
gfCNCPoint1[8403] = {X 72.5133, Y 40.2675, Z -1.3333, A 0.000, B 0.000, C 0.000 }
gfCNCPoint1[8404] = {X 73.3582, Y 40.7692, Z -1.3333, A 0.000, B 0.000, C 0.000 }
gfCNCPoint1[8405] = {X 74.0679, Y 41.4489, Z -1.3333, A 0.000, B 0.000, C 0.000 }
gfCNCPoint1[8406] = {X 74.6056, Y 42.2713, Z -1.3333, A 0.000, B 0.000, C 0.000 }
gfCNCPoint1[8407] = {X 74.9436, Y 43.1940, Z -1.3333, A 0.000, B 0.000, C 0.000 }
gfCNCPoint1[8408] = {X 75.0643, Y 44.1692, Z -1.3333, A 0.000, B 0.000, C 0.000 }
gfCNCPoint1[8409] = {X 75.0645, Y 45.0000, Z -1.3333, A 0.000, B 0.000, C 0.000 }
gfCNCPoint1[8410] = {X 74.9561, Y 45.9613, Z -1.3333, A 0.000, B 0.000, C 0.000 }
gfCNCPoint1[8411] = {X 74.6366, Y 46.8744, Z -1.3333, A 0.000, B 0.000, C 0.000 }
gfCNCPoint1[8412] = {X 74.1220, Y 47.6935, Z -1.3333, A 0.000, B 0.000, C 0.000 }
gfCNCPoint1[8413] = {X 73.4379, Y 48.3775, Z -1.3333, A 0.000, B 0.000, C 0.000 }
gfCNCPoint1[8414] = {X 72.6188, Y 48.8922, Z -1.3333, A 0.000, B 0.000, C 0.000 }
gfCNCPoint1[8415] = {X 71.7057, Y 49.2117, Z -1.3333, A 0.000, B 0.000, C 0.000 }
gfCNCPoint1[8416] = {X 70.7445, Y 49.3200, Z -1.3333, A 0.000, B 0.000, C 0.000 }
gfCNCPoint1[8417] = {X 64.1851, Y 49.3200, Z -1.3333, A 0.000, B 0.000, C 0.000 }
gfCNCPoint1[8418] = {X 63.2238, Y 49.2117, Z -1.3333, A 0.000, B 0.000, C 0.000 }
gfCNCPoint1[8419] = {X 62.3108, Y 48.8922, Z -1.3333, A 0.000, B 0.000, C 0.000 }
gfCNCPoint1[8420] = {X 61.4917, Y 48.3775, Z -1.3333, A 0.000, B 0.000, C 0.000 }
gfCNCPoint1[8421] = {X 60.8076, Y 47.6935, Z -1.3333, A 0.000, B 0.000, C 0.000 }
gfCNCPoint1[8422] = {X 60.2929, Y 46.8744, Z -1.3333, A 0.000, B 0.000, C 0.000 }
gfCNCPoint1[8423] = {X 59.9734, Y 45.9613, Z -1.3333, A 0.000, B 0.000, C 0.000 }
gfCNCPoint1[8424] = {X 59.8651, Y 45.0000, Z -1.3333, A 0.000, B 0.000, C 0.000 }
gfCNCPoint1[8425] = {X 59.8651, Y 44.2084, Z -1.3333, A 0.000, B 0.000, C 0.000 }
gfCNCPoint1[8426] = {X 59.9522, Y 43.3499, Z -1.3333, A 0.000, B 0.000, C 0.000 }
gfCNCPoint1[8427] = {X 60.2081, Y 42.5258, Z -1.3333, A 0.000, B 0.000, C 0.000 }
gfCNCPoint1[8428] = {X 60.6227, Y 41.7690, Z -1.3333, A 0.000, B 0.000, C 0.000 }
gfCNCPoint1[8429] = {X 60.0075, Y 40.0892, Z -1.3333, A 0.000, B 0.000, C 0.000 }
gfCNCPoint1[8430] = {X 52.0762, Y 40.0892, Z -1.3333, A 0.000, B 0.000, C 0.000 }
gfCNCPoint1[8431] = {X 51.3337, Y 42.0835, Z -1.3333, A 0.000, B 0.000, C 0.000 }
gfCNCPoint1[8432] = {X 51.3370, Y 42.0888, Z -1.3333, A 0.000, B 0.000, C 0.000 }
gfCNCPoint1[8433] = {X 51.6387, Y 42.7486, Z -1.3333, A 0.000, B 0.000, C 0.000 }
gfCNCPoint1[8434] = {X 51.8257, Y 43.4496, Z -1.3333, A 0.000, B 0.000, C 0.000 }
gfCNCPoint1[8435] = {X 51.8928, Y 44.1720, Z -1.3333, A 0.000, B 0.000, C 0.000 }
gfCNCPoint1[8436] = {X 51.8929, Y 45.0000, Z -1.3333, A 0.000, B 0.000, C 0.000 }
gfCNCPoint1[8437] = {X 51.7846, Y 45.9613, Z -1.3333, A 0.000, B 0.000, C 0.000 }
gfCNCPoint1[8438] = {X 51.4651, Y 46.8744, Z -1.3333, A 0.000, B 0.000, C 0.000 }
gfCNCPoint1[8439] = {X 50.9504, Y 47.6935, Z -1.3333, A 0.000, B 0.000, C 0.000 }
gfCNCPoint1[8440] = {X 50.2664, Y 48.3775, Z -1.3333, A 0.000, B 0.000, C 0.000 }
gfCNCPoint1[8441] = {X 49.4473, Y 48.8922, Z -1.3333, A 0.000, B 0.000, C 0.000 }
gfCNCPoint1[8442] = {X 48.5342, Y 49.2117, Z -1.3333, A 0.000, B 0.000, C 0.000 }
gfCNCPoint1[8443] = {X 47.5729, Y 49.3200, Z -1.3333, A 0.000, B 0.000, C 0.000 }
gfCNCPoint1[8444] = {X 40.6393, Y 49.3200, Z -1.3333, A 0.000, B 0.000, C 0.000 }
gfCNCPoint1[8445] = {X 39.6780, Y 49.2117, Z -1.3333, A 0.000, B 0.000, C 0.000 }
gfCNCPoint1[8446] = {X 38.7649, Y 48.8922, Z -1.3333, A 0.000, B 0.000, C 0.000 }
gfCNCPoint1[8447] = {X 37.9458, Y 48.3775, Z -1.3333, A 0.000, B 0.000, C 0.000 }
gfCNCPoint1[8448] = {X 37.2618, Y 47.6935, Z -1.3333, A 0.000, B 0.000, C 0.000 }
gfCNCPoint1[8449] = {X 36.7471, Y 46.8744, Z -1.3333, A 0.000, B 0.000, C 0.000 }
gfCNCPoint1[8450] = {X 36.4276, Y 45.9613, Z -1.3333, A 0.000, B 0.000, C 0.000 }
gfCNCPoint1[8451] = {X 36.3193, Y 45.0000, Z -1.3333, A 0.000, B 0.000, C 0.000 }
gfCNCPoint1[8452] = {X 36.3193, Y 44.2086, Z -1.3333, A 0.000, B 0.000, C 0.000 }
gfCNCPoint1[8453] = {X 36.4361, Y 43.2113, Z -1.3333, A 0.000, B 0.000, C 0.000 }
gfCNCPoint1[8454] = {X 36.7801, Y 42.2678, Z -1.3333, A 0.000, B 0.000, C 0.000 }
gfCNCPoint1[8455] = {X 37.3326, Y 41.4292, Z -1.3333, A 0.000, B 0.000, C 0.000 }
gfCNCPoint1[8456] = {X 38.0638, Y 40.7409, Z -1.3333, A 0.000, B 0.000, C 0.000 }
gfCNCPoint1[8457] = {X 38.9341, Y 40.2400, Z -1.3333, A 0.000, B 0.000, C 0.000 }
gfCNCPoint1[8458] = {X 39.5245, Y 38.8445, Z -1.3333, A 0.000, B 0.000, C 0.000 }
gfCNCPoint1[8459] = {X 40.0657, Y 37.4292, Z -1.3333, A 0.000, B 0.000, C 0.000 }
gfCNCPoint1[8460] = {X 43.6491, Y 27.8070, Z -1.3333, A 0.000, B 0.000, C 0.000 }
gfCNCPoint1[8461] = {X 39.9006, Y 26.4110, Z -1.3333, A 0.000, B 0.000, C 0.000 }
gfCNCPoint1[8462] = {X 43.7241, Y 27.8349, Z -1.3333, A 0.000, B 0.000, C 0.000 }
gfCNCPoint1[8463] = {X 48.3793, Y 15.3344, Z -1.3333, A 0.000, B 0.000, C 0.000 }
gfCNCPoint1[8464] = {X 47.9921, Y 14.6130, Z -1.3333, A 0.000, B 0.000, C 0.000 }
gfCNCPoint1[8465] = {X 47.7508, Y 13.8306, Z -1.3333, A 0.000, B 0.000, C 0.000 }
gfCNCPoint1[8466] = {X 47.6644, Y 13.0164, Z -1.3333, A 0.000, B 0.000, C 0.000 }
gfCNCPoint1[8467] = {X 47.6642, Y 12.1868, Z -1.3333, A 0.000, B 0.000, C 0.000 }
gfCNCPoint1[8468] = {X 47.7705, Y 11.2433, Z -1.3333, A 0.000, B 0.000, C 0.000 }
gfCNCPoint1[8469] = {X 48.0841, Y 10.3472, Z -1.3333, A 0.000, B 0.000, C 0.000 }
gfCNCPoint1[8470] = {X 48.5893, Y 9.5432, Z -1.3333, A 0.000, B 0.000, C 0.000 }
gfCNCPoint1[8471] = {X 49.2606, Y 8.8719, Z -1.3333, A 0.000, B 0.000, C 0.000 }
gfCNCPoint1[8472] = {X 50.0646, Y 8.3667, Z -1.3333, A 0.000, B 0.000, C 0.000 }
gfCNCPoint1[8473] = {X 50.9607, Y 8.0531, Z -1.3333, A 0.000, B 0.000, C 0.000 }
gfCNCPoint1[8474] = {X 51.9042, Y 7.9468, Z -1.3333, A 0.000, B 0.000, C 0.000 }
gfCNCPoint1[8475] = {X 59.6221, Y 7.9468, Z -1.3333, A 0.000, B 0.000, C 0.000 }
